LIN {X -0.049,Y -176.502,Z 1174.767,A 0.000,B 0.000,C 90.000,E1 138.162} C_DIS
LIN {X 0.075,Y -180.801,Z 1174.753,A 0.000,B 0.000,C 90.000,E1 135.567} C_DIS
LIN {X 0.061,Y -186.209,Z 1174.735,A 0.000,B 0.000,C 90.000,E1 132.204} C_DIS
LIN {X 0.000,Y -190.846,Z 1174.721,A 0.000,B 0.000,C 90.000,E1 129.725} C_DIS
LIN {X 0.034,Y -196.606,Z 1174.702,A 0.000,B 0.000,C 90.000,E1 126.423} C_DIS
LIN {X 0.006,Y -201.153,Z 1174.690,A 0.000,B 0.000,C 90.000,E1 124.119} C_DIS
LIN {X -0.026,Y -310.936,Z 1174.690,A 0.000,B 0.000,C 90.000,E1 124.119} C_DIS
LIN {X 0.002,Y -315.080,Z 1174.689,A 0.000,B 0.000,C 90.000,E1 123.992} C_DIS
LIN {X 0.113,Y -317.999,Z 1174.688,A 0.000,B 0.000,C 90.000,E1 123.785} C_DIS
LIN {X 0.000,Y -321.723,Z 1174.686,A 0.000,B 0.000,C 90.000,E1 123.420} C_DIS
LIN {X 0.084,Y -325.167,Z 1174.682,A 0.000,B 0.000,C 90.000,E1 122.832} C_DIS
LIN {X -0.013,Y -327.638,Z 1174.679,A 0.000,B 0.000,C 90.000,E1 122.212} C_DIS
LIN {X -0.136,Y -338.542,Z 1174.663,A 0.000,B 0.000,C 90.000,E1 119.411} C_DIS
LIN {X 0.016,Y -350.831,Z 1174.648,A 0.000,B 0.000,C 90.000,E1 116.616} C_DIS
LIN {X 0.063,Y -364.604,Z 1174.633,A 0.000,B 0.000,C 90.000,E1 113.898} C_DIS
LIN {X 0.100,Y -378.196,Z 1174.620,A 0.000,B 0.000,C 90.000,E1 111.535} C_DIS
LIN {X -0.165,Y -393.156,Z 1174.607,A 0.000,B 0.000,C 90.000,E1 109.268} C_DIS
LIN {X 0.055,Y -409.587,Z 1174.594,A 0.000,B 0.000,C 90.000,E1 106.985} C_DIS
LIN {X 0.182,Y -427.609,Z 1174.582,A 0.000,B 0.000,C 90.000,E1 104.773} C_DIS
LIN {X 0.246,Y -447.177,Z 1174.570,A 0.000,B 0.000,C 90.000,E1 102.647} C_DIS
LIN {X -0.025,Y -470.021,Z 1174.558,A 0.000,B 0.000,C 90.000,E1 100.489} C_DIS
LIN {X -0.016,Y -472.082,Z 1174.557,A 0.000,B 0.000,C 90.000,E1 100.254} C_DIS
LIN {X -0.007,Y -473.647,Z 1174.556,A 0.000,B 0.000,C 90.000,E1 100.018} C_DIS
LIN {X -0.147,Y -474.925,Z 1174.554,A 0.000,B 0.000,C 90.000,E1 99.782} C_DIS
LIN {X 0.101,Y -475.866,Z 1174.553,A 0.000,B 0.000,C 90.000,E1 99.500} C_DIS
LIN {X -0.166,Y -476.904,Z 1174.550,A 0.000,B 0.000,C 90.000,E1 99.029} C_DIS
LIN {X -0.033,Y -476.952,Z 1174.547,A 0.000,B 0.000,C 90.000,E1 98.511} C_DIS
LIN {X 0.109,Y -476.021,Z 1174.544,A 0.000,B 0.000,C 90.000,E1 97.992} C_DIS
LIN {X -0.219,Y -473.955,Z 1174.542,A 0.000,B 0.000,C 90.000,E1 97.530} C_DIS
LIN {X 0.115,Y -472.362,Z 1174.540,A 0.000,B 0.000,C 90.000,E1 97.239} C_DIS
LIN {X 0.027,Y -457.874,Z 1174.529,A 0.000,B 0.000,C 90.000,E1 95.220} C_DIS
LIN {X -0.055,Y -440.340,Z 1174.515,A 0.000,B 0.000,C 90.000,E1 92.636} C_DIS
LIN {X -0.091,Y -422.563,Z 1174.498,A 0.000,B 0.000,C 90.000,E1 89.714} C_DIS
LIN {X -0.002,Y -409.192,Z 1174.485,A 0.000,B 0.000,C 90.000,E1 87.249} C_DIS
LIN {X 0.069,Y -398.908,Z 1174.474,A 0.000,B 0.000,C 90.000,E1 85.298} C_DIS
LIN {X 0.035,Y -385.631,Z 1174.460,A 0.000,B 0.000,C 90.000,E1 82.761} C_DIS
LIN {X 0.104,Y -376.810,Z 1174.450,A 0.000,B 0.000,C 90.000,E1 81.027} C_DIS
LIN {X 0.065,Y -367.674,Z 1174.441,A 0.000,B 0.000,C 90.000,E1 79.285} C_DIS
LIN {X 0.006,Y -358.241,Z 1174.431,A 0.000,B 0.000,C 90.000,E1 77.521} C_DIS
LIN {X 0.129,Y -348.588,Z 1174.421,A 0.000,B 0.000,C 90.000,E1 75.700} C_DIS
LIN {X 0.145,Y -337.276,Z 1174.409,A 0.000,B 0.000,C 90.000,E1 73.559} C_DIS
LIN {X -0.024,Y -324.592,Z 1174.395,A 0.000,B 0.000,C 90.000,E1 71.094} C_DIS
LIN {X -0.063,Y -310.987,Z 1174.379,A 0.000,B 0.000,C 90.000,E1 68.230} C_DIS
LIN {X -0.001,Y -298.149,Z 1174.363,A 0.000,B 0.000,C 90.000,E1 65.281} C_DIS
LIN {X -0.038,Y -286.076,Z 1174.346,A 0.000,B 0.000,C 90.000,E1 62.281} C_DIS
LIN {X -0.066,Y -273.394,Z 1174.327,A 0.000,B 0.000,C 90.000,E1 58.869} C_DIS
LIN {X -0.117,Y -263.733,Z 1174.311,A 0.000,B 0.000,C 90.000,E1 56.087} C_DIS
LIN {X 0.091,Y -252.281,Z 1174.292,A 0.000,B 0.000,C 90.000,E1 52.477} C_DIS
LIN {X 0.027,Y -242.627,Z 1174.273,A 0.000,B 0.000,C 90.000,E1 49.218} C_DIS
LIN {X 0.132,Y -232.705,Z 1174.253,A 0.000,B 0.000,C 90.000,E1 45.486} C_DIS
LIN {X -0.074,Y -223.677,Z 1174.232,A 0.000,B 0.000,C 90.000,E1 41.757} C_DIS
LIN {X -0.011,Y -215.431,Z 1174.210,A 0.000,B 0.000,C 90.000,E1 37.890} C_DIS
LIN {X -0.081,Y -207.948,Z 1174.189,A 0.000,B 0.000,C 90.000,E1 33.992} C_DIS
LIN {X -0.038,Y -201.142,Z 1174.167,A 0.000,B 0.000,C 90.000,E1 30.001} C_DIS
LIN {X -0.083,Y -195.095,Z 1174.144,A 0.000,B 0.000,C 90.000,E1 25.976} C_DIS
LIN {X 0.054,Y -189.968,Z 1174.121,A 0.000,B 0.000,C 90.000,E1 21.844} C_DIS
LIN {X 0.099,Y -185.676,Z 1174.099,A 0.000,B 0.000,C 90.000,E1 17.692} C_DIS
LIN {X 0.036,Y -182.382,Z 1174.075,A 0.000,B 0.000,C 90.000,E1 13.536} C_DIS
LIN {X 0.030,Y -179.396,Z 1174.042,A 0.000,B 0.000,C 90.000,E1 7.644} C_DIS
LIN {X 0.062,Y -180.217,Z 1173.969,A 0.000,B 0.000,C 90.000,E1 354.432} C_DIS
LIN {X -0.014,Y -183.167,Z 1173.941,A 0.000,B 0.000,C 90.000,E1 349.398} C_DIS
LIN {X -0.066,Y -186.673,Z 1173.918,A 0.000,B 0.000,C 90.000,E1 345.227} C_DIS
LIN {X 0.052,Y -191.138,Z 1173.895,A 0.000,B 0.000,C 90.000,E1 341.040} C_DIS
LIN {X 0.086,Y -196.284,Z 1173.872,A 0.000,B 0.000,C 90.000,E1 336.922} C_DIS
LIN {X 0.053,Y -202.230,Z 1173.849,A 0.000,B 0.000,C 90.000,E1 332.871} C_DIS
LIN {X 0.040,Y -208.789,Z 1173.827,A 0.000,B 0.000,C 90.000,E1 328.869} C_DIS
LIN {X 0.135,Y -215.942,Z 1173.805,A 0.000,B 0.000,C 90.000,E1 324.895} C_DIS
LIN {X -0.029,Y -222.299,Z 1173.788,A 0.000,B 0.000,C 90.000,E1 321.823} C_DIS
LIN {X -0.113,Y -229.684,Z 1173.771,A 0.000,B 0.000,C 90.000,E1 318.771} C_DIS
LIN {X 0.104,Y -239.207,Z 1173.752,A 0.000,B 0.000,C 90.000,E1 315.324} C_DIS
LIN {X 0.104,Y -250.116,Z 1173.734,A 0.000,B 0.000,C 90.000,E1 312.000} C_DIS
LIN {X 0.109,Y -262.391,Z 1173.715,A 0.000,B 0.000,C 90.000,E1 308.749} C_DIS
LIN {X -0.068,Y -271.258,Z 1173.704,A 0.000,B 0.000,C 90.000,E1 306.664} C_DIS
LIN {X 0.145,Y -280.911,Z 1173.692,A 0.000,B 0.000,C 90.000,E1 304.532} C_DIS
LIN {X 0.075,Y -291.557,Z 1173.681,A 0.000,B 0.000,C 90.000,E1 302.498} C_DIS
LIN {X -0.160,Y -307.099,Z 1173.666,A 0.000,B 0.000,C 90.000,E1 299.873} C_DIS
LIN {X -0.040,Y -319.840,Z 1173.655,A 0.000,B 0.000,C 90.000,E1 297.897} C_DIS
LIN {X 0.071,Y -331.588,Z 1173.646,A 0.000,B 0.000,C 90.000,E1 296.283} C_DIS
LIN {X -0.064,Y -354.903,Z 1173.631,A 0.000,B 0.000,C 90.000,E1 293.567} C_DIS
LIN {X -0.085,Y -370.931,Z 1173.622,A 0.000,B 0.000,C 90.000,E1 291.897} C_DIS
LIN {X 0.197,Y -392.686,Z 1173.610,A 0.000,B 0.000,C 90.000,E1 289.812} C_DIS
LIN {X -0.061,Y -403.296,Z 1173.605,A 0.000,B 0.000,C 90.000,E1 288.852} C_DIS
LIN {X -0.119,Y -411.028,Z 1173.600,A 0.000,B 0.000,C 90.000,E1 288.109} C_DIS
LIN {X 0.117,Y -421.163,Z 1173.595,A 0.000,B 0.000,C 90.000,E1 287.040} C_DIS
LIN {X -0.004,Y -428.577,Z 1173.590,A 0.000,B 0.000,C 90.000,E1 286.260} C_DIS
LIN {X 0.222,Y -435.639,Z 1173.586,A 0.000,B 0.000,C 90.000,E1 285.426} C_DIS
LIN {X -0.038,Y -442.111,Z 1173.581,A 0.000,B 0.000,C 90.000,E1 284.662} C_DIS
LIN {X -0.141,Y -447.808,Z 1173.577,A 0.000,B 0.000,C 90.000,E1 283.883} C_DIS
LIN {X 0.141,Y -452.846,Z 1173.573,A 0.000,B 0.000,C 90.000,E1 283.063} C_DIS
LIN {X 0.025,Y -457.271,Z 1173.568,A 0.000,B 0.000,C 90.000,E1 282.299} C_DIS
LIN {X -0.050,Y -461.054,Z 1173.564,A 0.000,B 0.000,C 90.000,E1 281.535} C_DIS
LIN {X -0.188,Y -464.245,Z 1173.560,A 0.000,B 0.000,C 90.000,E1 280.782} C_DIS
LIN {X -0.051,Y -466.130,Z 1173.557,A 0.000,B 0.000,C 90.000,E1 280.254} C_DIS
LIN {X 0.089,Y -467.783,Z 1173.554,A 0.000,B 0.000,C 90.000,E1 279.726} C_DIS
LIN {X 0.163,Y -469.229,Z 1173.551,A 0.000,B 0.000,C 90.000,E1 279.208} C_DIS
LIN {X -0.216,Y -470.449,Z 1173.548,A 0.000,B 0.000,C 90.000,E1 278.746} C_DIS
LIN {X -0.051,Y -471.453,Z 1173.546,A 0.000,B 0.000,C 90.000,E1 278.219} C_DIS
LIN {X 0.053,Y -472.097,Z 1173.543,A 0.000,B 0.000,C 90.000,E1 277.701} C_DIS
LIN {X 0.163,Y -472.368,Z 1173.540,A 0.000,B 0.000,C 90.000,E1 277.182} C_DIS
LIN {X -0.191,Y -472.233,Z 1173.537,A 0.000,B 0.000,C 90.000,E1 276.720} C_DIS
LIN {X -0.073,Y -471.696,Z 1173.534,A 0.000,B 0.000,C 90.000,E1 276.201} C_DIS
LIN {X 0.043,Y -470.719,Z 1173.532,A 0.000,B 0.000,C 90.000,E1 275.682} C_DIS
LIN {X 0.155,Y -469.304,Z 1173.529,A 0.000,B 0.000,C 90.000,E1 275.163} C_DIS
LIN {X -0.208,Y -467.421,Z 1173.526,A 0.000,B 0.000,C 90.000,E1 274.702} C_DIS
LIN {X -0.149,Y -465.013,Z 1173.523,A 0.000,B 0.000,C 90.000,E1 274.188} C_DIS
LIN {X -0.071,Y -461.983,Z 1173.520,A 0.000,B 0.000,C 90.000,E1 273.669} C_DIS
LIN {X -0.039,Y -458.095,Z 1173.517,A 0.000,B 0.000,C 90.000,E1 273.154} C_DIS
LIN {X 0.220,Y -455.772,Z 1173.516,A 0.000,B 0.000,C 90.000,E1 272.865} C_DIS
LIN {X -0.138,Y -450.334,Z 1173.513,A 0.000,B 0.000,C 90.000,E1 272.407} C_DIS
LIN {X -0.112,Y -444.074,Z 1173.511,A 0.000,B 0.000,C 90.000,E1 271.949} C_DIS
LIN {X 0.025,Y -437.430,Z 1173.509,A 0.000,B 0.000,C 90.000,E1 271.547} C_DIS
LIN {X 0.201,Y -430.402,Z 1173.507,A 0.000,B 0.000,C 90.000,E1 271.203} C_DIS
LIN {X -0.067,Y -423.443,Z 1173.505,A 0.000,B 0.000,C 90.000,E1 270.974} C_DIS
LIN {X -0.032,Y -416.454,Z 1173.504,A 0.000,B 0.000,C 90.000,E1 270.745} C_DIS
LIN {X 0.056,Y -405.575,Z 1173.503,A 0.000,B 0.000,C 90.000,E1 270.458} C_DIS
LIN {X 0.138,Y -391.567,Z 1173.501,A 0.000,B 0.000,C 90.000,E1 270.172} C_DIS
LIN {X 0.102,Y -383.629,Z 1173.500,A 0.000,B 0.000,C 90.000,E1 270.057} C_DIS
LIN {X -0.178,Y -371.294,Z 1173.500,A 0.000,B 0.000,C 90.000,E1 270.000} C_DIS
LIN {X 0.140,Y -369.390,Z 1173.500,A 0.000,B 0.000,C 90.000,E1 269.943} C_DIS
LIN {X 0.044,Y -181.553,Z 1173.500,A 0.000,B 0.000,C 90.000,E1 269.943} C_DIS
LIN {X 0.055,Y -180.823,Z 1173.471,A 0.000,B 0.000,C 90.000,E1 264.837} C_DIS
LIN {X -0.044,Y -178.926,Z 1173.443,A 0.000,B 0.000,C 90.000,E1 259.803} C_DIS
LIN {X -0.006,Y -175.974,Z 1173.415,A 0.000,B 0.000,C 90.000,E1 254.700} C_DIS
LIN {X -0.061,Y -175.460,Z 1173.410,A 0.000,B 0.000,C 90.000,E1 253.866} C_DIS
LIN {X -0.004,Y -172.211,Z 1173.386,A 0.000,B 0.000,C 90.000,E1 249.571} C_DIS
LIN {X -0.026,Y -171.686,Z 1173.382,A 0.000,B 0.000,C 90.000,E1 248.720} C_DIS
LIN {X -0.035,Y -167.913,Z 1173.358,A 0.000,B 0.000,C 90.000,E1 244.409} C_DIS
LIN {X -0.017,Y -166.655,Z 1173.348,A 0.000,B 0.000,C 90.000,E1 242.666} C_DIS
LIN {X 0.038,Y -162.638,Z 1173.324,A 0.000,B 0.000,C 90.000,E1 238.280} C_DIS
LIN {X -0.038,Y -161.326,Z 1173.314,A 0.000,B 0.000,C 90.000,E1 236.548} C_DIS
LIN {X 0.005,Y -157.322,Z 1173.290,A 0.000,B 0.000,C 90.000,E1 232.110} C_DIS
LIN {X -0.062,Y -155.303,Z 1173.275,A 0.000,B 0.000,C 90.000,E1 229.461} C_DIS
LIN {X 0.084,Y -151.662,Z 1173.250,A 0.000,B 0.000,C 90.000,E1 224.919} C_DIS
LIN {X 0.021,Y -150.529,Z 1173.240,A 0.000,B 0.000,C 90.000,E1 223.137} C_DIS
LIN {X -0.048,Y -147.253,Z 1173.214,A 0.000,B 0.000,C 90.000,E1 218.624} C_DIS
LIN {X 0.008,Y -145.278,Z 1173.194,A 0.000,B 0.000,C 90.000,E1 214.945} C_DIS
LIN {X 0.042,Y -142.382,Z 1173.163,A 0.000,B 0.000,C 90.000,E1 209.411} C_DIS
LIN {X -0.035,Y -141.359,Z 1173.148,A 0.000,B 0.000,C 90.000,E1 206.668} C_DIS
LIN {X 0.074,Y -139.342,Z 1173.112,A 0.000,B 0.000,C 90.000,E1 200.120} C_DIS
LIN {X -0.051,Y -139.010,Z 1173.102,A 0.000,B 0.000,C 90.000,E1 198.308} C_DIS
LIN {X -0.056,Y -138.341,Z 1173.055,A 0.000,B 0.000,C 90.000,E1 189.905} C_DIS
LIN {X -0.036,Y -139.399,Z 1173.008,A 0.000,B 0.000,C 90.000,E1 181.489} C_DIS
LIN {X 0.017,Y -141.304,Z 1172.972,A 0.000,B 0.000,C 90.000,E1 174.951} C_DIS
LIN {X -0.025,Y -142.664,Z 1172.957,A 0.000,B 0.000,C 90.000,E1 172.186} C_DIS
LIN {X -0.076,Y -145.011,Z 1172.931,A 0.000,B 0.000,C 90.000,E1 167.589} C_DIS
LIN {X 0.055,Y -147.638,Z 1172.911,A 0.000,B 0.000,C 90.000,E1 163.866} C_DIS
LIN {X -0.009,Y -150.270,Z 1172.890,A 0.000,B 0.000,C 90.000,E1 160.242} C_DIS
LIN {X 0.004,Y -153.671,Z 1172.870,A 0.000,B 0.000,C 90.000,E1 156.613} C_DIS
LIN {X 0.061,Y -157.086,Z 1172.850,A 0.000,B 0.000,C 90.000,E1 152.999} C_DIS
LIN {X -0.002,Y -161.221,Z 1172.830,A 0.000,B 0.000,C 90.000,E1 149.459} C_DIS
LIN {X -0.054,Y -163.310,Z 1172.821,A 0.000,B 0.000,C 90.000,E1 147.709} C_DIS
LIN {X -0.044,Y -167.760,Z 1172.801,A 0.000,B 0.000,C 90.000,E1 144.196} C_DIS
LIN {X 0.108,Y -171.576,Z 1172.786,A 0.000,B 0.000,C 90.000,E1 141.537} C_DIS
LIN {X -0.092,Y -176.525,Z 1172.767,A 0.000,B 0.000,C 90.000,E1 138.162} C_DIS
LIN {X 0.032,Y -180.823,Z 1172.753,A 0.000,B 0.000,C 90.000,E1 135.567} C_DIS
LIN {X 0.017,Y -186.232,Z 1172.734,A 0.000,B 0.000,C 90.000,E1 132.204} C_DIS
LIN {X -0.045,Y -190.869,Z 1172.721,A 0.000,B 0.000,C 90.000,E1 129.725} C_DIS
LIN {X -0.012,Y -196.631,Z 1172.702,A 0.000,B 0.000,C 90.000,E1 126.423} C_DIS
LIN {X 0.079,Y -201.118,Z 1172.690,A 0.000,B 0.000,C 90.000,E1 124.119} C_DIS
LIN {X 0.086,Y -310.102,Z 1172.690,A 0.000,B 0.000,C 90.000,E1 124.119} C_DIS
LIN {X -0.070,Y -315.565,Z 1172.689,A 0.000,B 0.000,C 90.000,E1 123.992} C_DIS
LIN {X -0.063,Y -318.498,Z 1172.688,A 0.000,B 0.000,C 90.000,E1 123.785} C_DIS
LIN {X -0.088,Y -322.233,Z 1172.685,A 0.000,B 0.000,C 90.000,E1 123.372} C_DIS
LIN {X 0.086,Y -324.120,Z 1172.684,A 0.000,B 0.000,C 90.000,E1 123.038} C_DIS
LIN {X -0.013,Y -325.596,Z 1172.682,A 0.000,B 0.000,C 90.000,E1 122.752} C_DIS
LIN {X 0.078,Y -338.901,Z 1172.663,A 0.000,B 0.000,C 90.000,E1 119.283} C_DIS
LIN {X -0.065,Y -351.237,Z 1172.647,A 0.000,B 0.000,C 90.000,E1 116.539} C_DIS
LIN {X -0.018,Y -365.061,Z 1172.632,A 0.000,B 0.000,C 90.000,E1 113.823} C_DIS
LIN {X 0.020,Y -378.702,Z 1172.619,A 0.000,B 0.000,C 90.000,E1 111.461} C_DIS
LIN {X 0.126,Y -393.714,Z 1172.606,A 0.000,B 0.000,C 90.000,E1 109.141} C_DIS
LIN {X -0.024,Y -410.202,Z 1172.594,A 0.000,B 0.000,C 90.000,E1 106.913} C_DIS
LIN {X -0.005,Y -428.284,Z 1172.582,A 0.000,B 0.000,C 90.000,E1 104.717} C_DIS
LIN {X 0.092,Y -447.891,Z 1172.570,A 0.000,B 0.000,C 90.000,E1 102.591} C_DIS
LIN {X -0.043,Y -470.651,Z 1172.558,A 0.000,B 0.000,C 90.000,E1 100.423} C_DIS
LIN {X -0.166,Y -472.574,Z 1172.557,A 0.000,B 0.000,C 90.000,E1 100.197} C_DIS
LIN {X -0.204,Y -474.036,Z 1172.555,A 0.000,B 0.000,C 90.000,E1 99.962} C_DIS
LIN {X -0.093,Y -476.032,Z 1172.552,A 0.000,B 0.000,C 90.000,E1 99.443} C_DIS
LIN {X 0.106,Y -476.898,Z 1172.550,A 0.000,B 0.000,C 90.000,E1 98.916} C_DIS
LIN {X -0.230,Y -476.784,Z 1172.547,A 0.000,B 0.000,C 90.000,E1 98.454} C_DIS
LIN {X -0.088,Y -475.679,Z 1172.544,A 0.000,B 0.000,C 90.000,E1 97.936} C_DIS
LIN {X -0.219,Y -474.704,Z 1172.543,A 0.000,B 0.000,C 90.000,E1 97.701} C_DIS
LIN {X 0.118,Y -473.387,Z 1172.541,A 0.000,B 0.000,C 90.000,E1 97.409} C_DIS
LIN {X 0.045,Y -458.988,Z 1172.530,A 0.000,B 0.000,C 90.000,E1 95.391} C_DIS
LIN {X -0.012,Y -441.392,Z 1172.516,A 0.000,B 0.000,C 90.000,E1 92.808} C_DIS
LIN {X 0.103,Y -421.988,Z 1172.498,A 0.000,B 0.000,C 90.000,E1 89.599} C_DIS
LIN {X 0.170,Y -408.639,Z 1172.484,A 0.000,B 0.000,C 90.000,E1 87.135} C_DIS
LIN {X -0.174,Y -398.345,Z 1172.473,A 0.000,B 0.000,C 90.000,E1 85.241} C_DIS
LIN {X 0.166,Y -385.048,Z 1172.459,A 0.000,B 0.000,C 90.000,E1 82.648} C_DIS
LIN {X -0.154,Y -376.199,Z 1172.450,A 0.000,B 0.000,C 90.000,E1 80.971} C_DIS
LIN {X -0.130,Y -367.052,Z 1172.440,A 0.000,B 0.000,C 90.000,E1 79.218} C_DIS
LIN {X 0.085,Y -357.601,Z 1172.430,A 0.000,B 0.000,C 90.000,E1 77.409} C_DIS
LIN {X -0.149,Y -347.926,Z 1172.420,A 0.000,B 0.000,C 90.000,E1 75.644} C_DIS
LIN {X 0.167,Y -334.992,Z 1172.406,A 0.000,B 0.000,C 90.000,E1 73.142} C_DIS
LIN {X -0.059,Y -322.397,Z 1172.393,A 0.000,B 0.000,C 90.000,E1 70.678} C_DIS
LIN {X 0.183,Y -306.046,Z 1172.373,A 0.000,B 0.000,C 90.000,E1 67.102} C_DIS
LIN {X -0.031,Y -292.134,Z 1172.355,A 0.000,B 0.000,C 90.000,E1 63.845} C_DIS
LIN {X 0.019,Y -280.314,Z 1172.338,A 0.000,B 0.000,C 90.000,E1 60.795} C_DIS
LIN {X -0.072,Y -269.159,Z 1172.321,A 0.000,B 0.000,C 90.000,E1 57.709} C_DIS
LIN {X -0.033,Y -258.483,Z 1172.303,A 0.000,B 0.000,C 90.000,E1 54.529} C_DIS
LIN {X -0.045,Y -248.425,Z 1172.285,A 0.000,B 0.000,C 90.000,E1 51.295} C_DIS
LIN {X -0.059,Y -238.057,Z 1172.265,A 0.000,B 0.000,C 90.000,E1 47.634} C_DIS
LIN {X 0.055,Y -228.506,Z 1172.244,A 0.000,B 0.000,C 90.000,E1 43.866} C_DIS
LIN {X -0.097,Y -219.812,Z 1172.223,A 0.000,B 0.000,C 90.000,E1 40.092} C_DIS
LIN {X 0.052,Y -211.901,Z 1172.201,A 0.000,B 0.000,C 90.000,E1 36.171} C_DIS
LIN {X 0.092,Y -204.686,Z 1172.179,A 0.000,B 0.000,C 90.000,E1 32.212} C_DIS
LIN {X -0.005,Y -198.166,Z 1172.157,A 0.000,B 0.000,C 90.000,E1 28.231} C_DIS
LIN {X 0.035,Y -192.459,Z 1172.134,A 0.000,B 0.000,C 90.000,E1 24.155} C_DIS
LIN {X -0.053,Y -187.661,Z 1172.111,A 0.000,B 0.000,C 90.000,E1 20.066} C_DIS
LIN {X -0.020,Y -183.796,Z 1172.088,A 0.000,B 0.000,C 90.000,E1 15.898} C_DIS
LIN {X 0.062,Y -180.484,Z 1172.060,A 0.000,B 0.000,C 90.000,E1 10.838} C_DIS
LIN {X 0.063,Y -178.329,Z 1172.023,A 0.000,B 0.000,C 90.000,E1 4.073} C_DIS
LIN {X 0.050,Y -179.888,Z 1171.969,A 0.000,B 0.000,C 90.000,E1 354.432} C_DIS
LIN {X -0.038,Y -182.831,Z 1171.941,A 0.000,B 0.000,C 90.000,E1 349.398} C_DIS
LIN {X 0.079,Y -186.309,Z 1171.918,A 0.000,B 0.000,C 90.000,E1 345.172} C_DIS
LIN {X 0.004,Y -190.771,Z 1171.895,A 0.000,B 0.000,C 90.000,E1 341.040} C_DIS
LIN {X 0.024,Y -195.923,Z 1171.872,A 0.000,B 0.000,C 90.000,E1 336.922} C_DIS
LIN {X -0.020,Y -201.848,Z 1171.849,A 0.000,B 0.000,C 90.000,E1 332.871} C_DIS
LIN {X -0.050,Y -208.422,Z 1171.827,A 0.000,B 0.000,C 90.000,E1 328.869} C_DIS
LIN {X 0.031,Y -215.610,Z 1171.805,A 0.000,B 0.000,C 90.000,E1 324.895} C_DIS
LIN {X 0.030,Y -222.026,Z 1171.788,A 0.000,B 0.000,C 90.000,E1 321.778} C_DIS
LIN {X 0.086,Y -229.469,Z 1171.771,A 0.000,B 0.000,C 90.000,E1 318.690} C_DIS
LIN {X -0.033,Y -239.035,Z 1171.752,A 0.000,B 0.000,C 90.000,E1 315.324} C_DIS
LIN {X -0.044,Y -249.981,Z 1171.733,A 0.000,B 0.000,C 90.000,E1 312.000} C_DIS
LIN {X -0.050,Y -262.317,Z 1171.715,A 0.000,B 0.000,C 90.000,E1 308.749} C_DIS
LIN {X 0.146,Y -271.213,Z 1171.703,A 0.000,B 0.000,C 90.000,E1 306.583} C_DIS
LIN {X -0.083,Y -282.636,Z 1171.690,A 0.000,B 0.000,C 90.000,E1 304.199} C_DIS
LIN {X 0.032,Y -293.524,Z 1171.679,A 0.000,B 0.000,C 90.000,E1 302.133} C_DIS
LIN {X 0.074,Y -307.185,Z 1171.666,A 0.000,B 0.000,C 90.000,E1 299.795} C_DIS
LIN {X 0.052,Y -319.953,Z 1171.655,A 0.000,B 0.000,C 90.000,E1 297.847} C_DIS
LIN {X 0.172,Y -331.725,Z 1171.646,A 0.000,B 0.000,C 90.000,E1 296.232} C_DIS
LIN {X 0.092,Y -352.148,Z 1171.632,A 0.000,B 0.000,C 90.000,E1 293.823} C_DIS
LIN {X 0.011,Y -367.983,Z 1171.623,A 0.000,B 0.000,C 90.000,E1 292.153} C_DIS
LIN {X -0.135,Y -389.737,Z 1171.612,A 0.000,B 0.000,C 90.000,E1 290.120} C_DIS
LIN {X 0.151,Y -400.402,Z 1171.606,A 0.000,B 0.000,C 90.000,E1 289.087} C_DIS
LIN {X -0.083,Y -408.312,Z 1171.602,A 0.000,B 0.000,C 90.000,E1 288.362} C_DIS
LIN {X -0.057,Y -418.508,Z 1171.596,A 0.000,B 0.000,C 90.000,E1 287.330} C_DIS
LIN {X 0.051,Y -428.488,Z 1171.590,A 0.000,B 0.000,C 90.000,E1 286.260} C_DIS
LIN {X -0.141,Y -435.570,Z 1171.586,A 0.000,B 0.000,C 90.000,E1 285.481} C_DIS
LIN {X 0.019,Y -442.041,Z 1171.581,A 0.000,B 0.000,C 90.000,E1 284.662} C_DIS
LIN {X -0.085,Y -447.763,Z 1171.577,A 0.000,B 0.000,C 90.000,E1 283.883} C_DIS
LIN {X 0.198,Y -452.808,Z 1171.573,A 0.000,B 0.000,C 90.000,E1 283.063} C_DIS
LIN {X 0.081,Y -457.266,Z 1171.568,A 0.000,B 0.000,C 90.000,E1 282.299} C_DIS
LIN {X 0.007,Y -461.060,Z 1171.564,A 0.000,B 0.000,C 90.000,E1 281.535} C_DIS
LIN {X -0.131,Y -464.245,Z 1171.560,A 0.000,B 0.000,C 90.000,E1 280.782} C_DIS
LIN {X 0.007,Y -466.155,Z 1171.557,A 0.000,B 0.000,C 90.000,E1 280.254} C_DIS
LIN {X 0.147,Y -467.851,Z 1171.554,A 0.000,B 0.000,C 90.000,E1 279.726} C_DIS
LIN {X 0.221,Y -469.332,Z 1171.551,A 0.000,B 0.000,C 90.000,E1 279.208} C_DIS
LIN {X -0.156,Y -470.596,Z 1171.548,A 0.000,B 0.000,C 90.000,E1 278.746} C_DIS
LIN {X 0.009,Y -471.575,Z 1171.546,A 0.000,B 0.000,C 90.000,E1 278.219} C_DIS
LIN {X 0.113,Y -472.242,Z 1171.543,A 0.000,B 0.000,C 90.000,E1 277.701} C_DIS
LIN {X 0.225,Y -472.567,Z 1171.540,A 0.000,B 0.000,C 90.000,E1 277.182} C_DIS
LIN {X -0.128,Y -472.452,Z 1171.537,A 0.000,B 0.000,C 90.000,E1 276.720} C_DIS
LIN {X -0.010,Y -471.944,Z 1171.534,A 0.000,B 0.000,C 90.000,E1 276.201} C_DIS
LIN {X 0.107,Y -471.007,Z 1171.532,A 0.000,B 0.000,C 90.000,E1 275.682} C_DIS
LIN {X 0.220,Y -469.624,Z 1171.529,A 0.000,B 0.000,C 90.000,E1 275.163} C_DIS
LIN {X -0.142,Y -467.798,Z 1171.526,A 0.000,B 0.000,C 90.000,E1 274.702} C_DIS
LIN {X -0.080,Y -465.391,Z 1171.523,A 0.000,B 0.000,C 90.000,E1 274.188} C_DIS
LIN {X 0.000,Y -462.390,Z 1171.520,A 0.000,B 0.000,C 90.000,E1 273.669} C_DIS
LIN {X 0.034,Y -458.543,Z 1171.518,A 0.000,B 0.000,C 90.000,E1 273.154} C_DIS
LIN {X -0.163,Y -456.262,Z 1171.516,A 0.000,B 0.000,C 90.000,E1 272.922} C_DIS
LIN {X 0.073,Y -453.668,Z 1171.515,A 0.000,B 0.000,C 90.000,E1 272.636} C_DIS
LIN {X -0.084,Y -450.819,Z 1171.513,A 0.000,B 0.000,C 90.000,E1 272.407} C_DIS
LIN {X -0.109,Y -444.586,Z 1171.511,A 0.000,B 0.000,C 90.000,E1 271.949} C_DIS
LIN {X -0.022,Y -437.865,Z 1171.509,A 0.000,B 0.000,C 90.000,E1 271.547} C_DIS
LIN {X 0.119,Y -430.822,Z 1171.507,A 0.000,B 0.000,C 90.000,E1 271.203} C_DIS
LIN {X -0.163,Y -423.858,Z 1171.505,A 0.000,B 0.000,C 90.000,E1 270.974} C_DIS
LIN {X -0.112,Y -416.957,Z 1171.504,A 0.000,B 0.000,C 90.000,E1 270.745} C_DIS
LIN {X 0.188,Y -409.846,Z 1171.503,A 0.000,B 0.000,C 90.000,E1 270.516} C_DIS
LIN {X 0.174,Y -399.186,Z 1171.502,A 0.000,B 0.000,C 90.000,E1 270.286} C_DIS
LIN {X 0.049,Y -388.425,Z 1171.501,A 0.000,B 0.000,C 90.000,E1 270.115} C_DIS
LIN {X 0.083,Y -379.778,Z 1171.500,A 0.000,B 0.000,C 90.000,E1 270.000} C_DIS
LIN {X 0.080,Y -371.038,Z 1171.500,A 0.000,B 0.000,C 90.000,E1 269.943} C_DIS
LIN {X 0.026,Y -365.401,Z 1171.500,A 0.000,B 0.000,C 90.000,E1 269.943} C_DIS
LIN {X -0.013,Y -181.550,Z 1171.500,A 0.000,B 0.000,C 90.000,E1 269.943} C_DIS
LIN {X 0.021,Y -180.819,Z 1171.471,A 0.000,B 0.000,C 90.000,E1 264.837} C_DIS
LIN {X -0.078,Y -178.922,Z 1171.443,A 0.000,B 0.000,C 90.000,E1 259.803} C_DIS
LIN {X 0.006,Y -175.969,Z 1171.415,A 0.000,B 0.000,C 90.000,E1 254.685} C_DIS
LIN {X -0.046,Y -175.451,Z 1171.410,A 0.000,B 0.000,C 90.000,E1 253.850} C_DIS
LIN {X -0.037,Y -172.204,Z 1171.386,A 0.000,B 0.000,C 90.000,E1 249.571} C_DIS
LIN {X -0.059,Y -171.679,Z 1171.382,A 0.000,B 0.000,C 90.000,E1 248.720} C_DIS
LIN {X -0.068,Y -167.904,Z 1171.358,A 0.000,B 0.000,C 90.000,E1 244.409} C_DIS
LIN {X -0.050,Y -166.645,Z 1171.348,A 0.000,B 0.000,C 90.000,E1 242.666} C_DIS
LIN {X 0.005,Y -162.630,Z 1171.324,A 0.000,B 0.000,C 90.000,E1 238.280} C_DIS
LIN {X 0.064,Y -161.317,Z 1171.314,A 0.000,B 0.000,C 90.000,E1 236.501} C_DIS
LIN {X -0.026,Y -157.313,Z 1171.289,A 0.000,B 0.000,C 90.000,E1 232.110} C_DIS
LIN {X -0.093,Y -155.291,Z 1171.275,A 0.000,B 0.000,C 90.000,E1 229.461} C_DIS
LIN {X 0.053,Y -151.653,Z 1171.250,A 0.000,B 0.000,C 90.000,E1 224.919} C_DIS
LIN {X -0.010,Y -150.520,Z 1171.240,A 0.000,B 0.000,C 90.000,E1 223.137} C_DIS
LIN {X 0.014,Y -147.246,Z 1171.214,A 0.000,B 0.000,C 90.000,E1 218.588} C_DIS
LIN {X -0.022,Y -145.271,Z 1171.194,A 0.000,B 0.000,C 90.000,E1 214.945} C_DIS
LIN {X 0.012,Y -142.378,Z 1171.163,A 0.000,B 0.000,C 90.000,E1 209.411} C_DIS
LIN {X 0.062,Y -141.354,Z 1171.148,A 0.000,B 0.000,C 90.000,E1 206.616} C_DIS
LIN {X 0.045,Y -139.340,Z 1171.112,A 0.000,B 0.000,C 90.000,E1 200.120} C_DIS
LIN {X -0.036,Y -139.007,Z 1171.102,A 0.000,B 0.000,C 90.000,E1 198.290} C_DIS
LIN {X 0.051,Y -138.339,Z 1171.055,A 0.000,B 0.000,C 90.000,E1 189.849} C_DIS
LIN {X -0.065,Y -139.402,Z 1171.008,A 0.000,B 0.000,C 90.000,E1 181.489} C_DIS
LIN {X -0.012,Y -141.308,Z 1170.972,A 0.000,B 0.000,C 90.000,E1 174.951} C_DIS
LIN {X -0.055,Y -142.669,Z 1170.956,A 0.000,B 0.000,C 90.000,E1 172.186} C_DIS
LIN {X 0.067,Y -145.019,Z 1170.931,A 0.000,B 0.000,C 90.000,E1 167.521} C_DIS
LIN {X 0.025,Y -147.645,Z 1170.910,A 0.000,B 0.000,C 90.000,E1 163.866} C_DIS
LIN {X -0.040,Y -150.280,Z 1170.890,A 0.000,B 0.000,C 90.000,E1 160.242} C_DIS
LIN {X -0.027,Y -153.683,Z 1170.870,A 0.000,B 0.000,C 90.000,E1 156.613} C_DIS
LIN {X 0.028,Y -157.097,Z 1170.850,A 0.000,B 0.000,C 90.000,E1 152.999} C_DIS
LIN {X -0.033,Y -161.236,Z 1170.830,A 0.000,B 0.000,C 90.000,E1 149.459} C_DIS
LIN {X 0.052,Y -163.323,Z 1170.820,A 0.000,B 0.000,C 90.000,E1 147.661} C_DIS
LIN {X -0.077,Y -167.776,Z 1170.801,A 0.000,B 0.000,C 90.000,E1 144.196} C_DIS
LIN {X 0.075,Y -171.591,Z 1170.786,A 0.000,B 0.000,C 90.000,E1 141.537} C_DIS
LIN {X 0.005,Y -176.542,Z 1170.767,A 0.000,B 0.000,C 90.000,E1 138.119} C_DIS
LIN {X -0.002,Y -180.841,Z 1170.753,A 0.000,B 0.000,C 90.000,E1 135.567} C_DIS
LIN {X -0.018,Y -186.251,Z 1170.734,A 0.000,B 0.000,C 90.000,E1 132.204} C_DIS
LIN {X -0.080,Y -190.888,Z 1170.721,A 0.000,B 0.000,C 90.000,E1 129.725} C_DIS
LIN {X -0.048,Y -196.652,Z 1170.702,A 0.000,B 0.000,C 90.000,E1 126.423} C_DIS
LIN {X 0.114,Y -201.102,Z 1170.690,A 0.000,B 0.000,C 90.000,E1 124.119} C_DIS
LIN {X 0.141,Y -310.674,Z 1170.690,A 0.000,B 0.000,C 90.000,E1 124.119} C_DIS
LIN {X -0.128,Y -315.930,Z 1170.689,A 0.000,B 0.000,C 90.000,E1 123.992} C_DIS
LIN {X -0.154,Y -318.773,Z 1170.688,A 0.000,B 0.000,C 90.000,E1 123.785} C_DIS
LIN {X 0.145,Y -322.523,Z 1170.685,A 0.000,B 0.000,C 90.000,E1 123.293} C_DIS
LIN {X -0.010,Y -324.382,Z 1170.683,A 0.000,B 0.000,C 90.000,E1 123.007} C_DIS
LIN {X 0.106,Y -325.830,Z 1170.682,A 0.000,B 0.000,C 90.000,E1 122.673} C_DIS
LIN {X 0.062,Y -337.833,Z 1170.664,A 0.000,B 0.000,C 90.000,E1 119.539} C_DIS
LIN {X -0.109,Y -350.034,Z 1170.649,A 0.000,B 0.000,C 90.000,E1 116.796} C_DIS
LIN {X -0.102,Y -363.722,Z 1170.634,A 0.000,B 0.000,C 90.000,E1 114.079} C_DIS
LIN {X -0.098,Y -377.229,Z 1170.621,A 0.000,B 0.000,C 90.000,E1 111.716} C_DIS
LIN {X -0.027,Y -392.096,Z 1170.608,A 0.000,B 0.000,C 90.000,E1 109.396} C_DIS
LIN {X -0.094,Y -408.429,Z 1170.595,A 0.000,B 0.000,C 90.000,E1 107.149} C_DIS
LIN {X -0.125,Y -426.344,Z 1170.583,A 0.000,B 0.000,C 90.000,E1 104.954} C_DIS
LIN {X -0.137,Y -445.841,Z 1170.571,A 0.000,B 0.000,C 90.000,E1 102.827} C_DIS
LIN {X 0.024,Y -466.091,Z 1170.560,A 0.000,B 0.000,C 90.000,E1 100.838} C_DIS
LIN {X 0.067,Y -470.996,Z 1170.558,A 0.000,B 0.000,C 90.000,E1 100.366} C_DIS
LIN {X -0.105,Y -472.854,Z 1170.556,A 0.000,B 0.000,C 90.000,E1 100.141} C_DIS
LIN {X -0.193,Y -474.259,Z 1170.555,A 0.000,B 0.000,C 90.000,E1 99.905} C_DIS
LIN {X -0.002,Y -476.105,Z 1170.552,A 0.000,B 0.000,C 90.000,E1 99.378} C_DIS
LIN {X 0.121,Y -476.851,Z 1170.549,A 0.000,B 0.000,C 90.000,E1 98.859} C_DIS
LIN {X -0.214,Y -476.623,Z 1170.547,A 0.000,B 0.000,C 90.000,E1 98.398} C_DIS
LIN {X -0.005,Y -475.392,Z 1170.544,A 0.000,B 0.000,C 90.000,E1 97.871} C_DIS
LIN {X -0.203,Y -474.342,Z 1170.542,A 0.000,B 0.000,C 90.000,E1 97.644} C_DIS
LIN {X 0.133,Y -472.933,Z 1170.541,A 0.000,B 0.000,C 90.000,E1 97.352} C_DIS
LIN {X -0.176,Y -456.685,Z 1170.528,A 0.000,B 0.000,C 90.000,E1 95.106} C_DIS
LIN {X -0.019,Y -440.933,Z 1170.515,A 0.000,B 0.000,C 90.000,E1 92.751} C_DIS
LIN {X 0.082,Y -421.567,Z 1170.498,A 0.000,B 0.000,C 90.000,E1 89.542} C_DIS
LIN {X 0.138,Y -408.240,Z 1170.484,A 0.000,B 0.000,C 90.000,E1 87.078} C_DIS
LIN {X -0.180,Y -397.914,Z 1170.473,A 0.000,B 0.000,C 90.000,E1 85.179} C_DIS
LIN {X 0.114,Y -384.625,Z 1170.459,A 0.000,B 0.000,C 90.000,E1 82.591} C_DIS
LIN {X -0.154,Y -375.757,Z 1170.449,A 0.000,B 0.000,C 90.000,E1 80.905} C_DIS
LIN {X 0.162,Y -366.591,Z 1170.440,A 0.000,B 0.000,C 90.000,E1 79.106} C_DIS
LIN {X 0.008,Y -357.133,Z 1170.430,A 0.000,B 0.000,C 90.000,E1 77.353} C_DIS
LIN {X 0.188,Y -347.417,Z 1170.420,A 0.000,B 0.000,C 90.000,E1 75.519} C_DIS
LIN {X 0.069,Y -334.515,Z 1170.406,A 0.000,B 0.000,C 90.000,E1 73.087} C_DIS
LIN {X -0.063,Y -321.905,Z 1170.392,A 0.000,B 0.000,C 90.000,E1 70.604} C_DIS
LIN {X 0.055,Y -305.580,Z 1170.373,A 0.000,B 0.000,C 90.000,E1 67.050} C_DIS
LIN {X -0.045,Y -291.705,Z 1170.354,A 0.000,B 0.000,C 90.000,E1 63.768} C_DIS
LIN {X 0.000,Y -279.882,Z 1170.337,A 0.000,B 0.000,C 90.000,E1 60.717} C_DIS
LIN {X 0.054,Y -269.948,Z 1170.322,A 0.000,B 0.000,C 90.000,E1 57.946} C_DIS
LIN {X 0.145,Y -258.036,Z 1170.302,A 0.000,B 0.000,C 90.000,E1 54.402} C_DIS
LIN {X 0.108,Y -247.984,Z 1170.284,A 0.000,B 0.000,C 90.000,E1 51.170} C_DIS
LIN {X -0.109,Y -237.643,Z 1170.264,A 0.000,B 0.000,C 90.000,E1 47.553} C_DIS
LIN {X -0.005,Y -228.105,Z 1170.243,A 0.000,B 0.000,C 90.000,E1 43.785} C_DIS
LIN {X 0.000,Y -219.427,Z 1170.222,A 0.000,B 0.000,C 90.000,E1 39.967} C_DIS
LIN {X -0.032,Y -211.500,Z 1170.200,A 0.000,B 0.000,C 90.000,E1 36.091} C_DIS
LIN {X -0.004,Y -204.282,Z 1170.178,A 0.000,B 0.000,C 90.000,E1 32.133} C_DIS
LIN {X 0.060,Y -197.743,Z 1170.156,A 0.000,B 0.000,C 90.000,E1 28.103} C_DIS
LIN {X -0.091,Y -192.042,Z 1170.134,A 0.000,B 0.000,C 90.000,E1 24.079} C_DIS
LIN {X -0.020,Y -187.251,Z 1170.111,A 0.000,B 0.000,C 90.000,E1 19.939} C_DIS
LIN {X -0.054,Y -183.414,Z 1170.088,A 0.000,B 0.000,C 90.000,E1 15.788} C_DIS
LIN {X 0.055,Y -180.117,Z 1170.060,A 0.000,B 0.000,C 90.000,E1 10.715} C_DIS
LIN {X -0.031,Y -178.113,Z 1170.027,A 0.000,B 0.000,C 90.000,E1 4.821} C_DIS
LIN {X 0.038,Y -179.552,Z 1169.969,A 0.000,B 0.000,C 90.000,E1 354.432} C_DIS
LIN {X -0.063,Y -182.493,Z 1169.941,A 0.000,B 0.000,C 90.000,E1 349.398} C_DIS
LIN {X 0.043,Y -185.966,Z 1169.918,A 0.000,B 0.000,C 90.000,E1 345.172} C_DIS
LIN {X -0.043,Y -190.404,Z 1169.895,A 0.000,B 0.000,C 90.000,E1 341.040} C_DIS
LIN {X -0.035,Y -195.561,Z 1169.872,A 0.000,B 0.000,C 90.000,E1 336.922} C_DIS
LIN {X -0.094,Y -201.464,Z 1169.849,A 0.000,B 0.000,C 90.000,E1 332.871} C_DIS
LIN {X 0.040,Y -208.054,Z 1169.827,A 0.000,B 0.000,C 90.000,E1 328.820} C_DIS
LIN {X -0.072,Y -215.283,Z 1169.805,A 0.000,B 0.000,C 90.000,E1 324.895} C_DIS
LIN {X 0.053,Y -221.744,Z 1169.788,A 0.000,B 0.000,C 90.000,E1 321.743} C_DIS
LIN {X -0.040,Y -229.242,Z 1169.770,A 0.000,B 0.000,C 90.000,E1 318.690} C_DIS
LIN {X 0.001,Y -238.855,Z 1169.752,A 0.000,B 0.000,C 90.000,E1 315.283} C_DIS
LIN {X -0.006,Y -248.554,Z 1169.735,A 0.000,B 0.000,C 90.000,E1 312.324} C_DIS
LIN {X -0.049,Y -260.811,Z 1169.717,A 0.000,B 0.000,C 90.000,E1 309.072} C_DIS
LIN {X -0.019,Y -271.183,Z 1169.703,A 0.000,B 0.000,C 90.000,E1 306.583} C_DIS
LIN {X 0.137,Y -282.656,Z 1169.690,A 0.000,B 0.000,C 90.000,E1 304.119} C_DIS
LIN {X 0.085,Y -297.398,Z 1169.675,A 0.000,B 0.000,C 90.000,E1 301.416} C_DIS
LIN {X -0.086,Y -309.358,Z 1169.664,A 0.000,B 0.000,C 90.000,E1 299.461} C_DIS
LIN {X -0.139,Y -320.066,Z 1169.655,A 0.000,B 0.000,C 90.000,E1 297.847} C_DIS
LIN {X -0.024,Y -331.857,Z 1169.646,A 0.000,B 0.000,C 90.000,E1 296.232} C_DIS
LIN {X 0.004,Y -352.520,Z 1169.632,A 0.000,B 0.000,C 90.000,E1 293.770} C_DIS
LIN {X 0.077,Y -368.406,Z 1169.623,A 0.000,B 0.000,C 90.000,E1 292.078} C_DIS
LIN {X -0.083,Y -390.114,Z 1169.611,A 0.000,B 0.000,C 90.000,E1 290.066} C_DIS
LIN {X -0.171,Y -400.785,Z 1169.606,A 0.000,B 0.000,C 90.000,E1 289.087} C_DIS
LIN {X -0.036,Y -408.711,Z 1169.602,A 0.000,B 0.000,C 90.000,E1 288.308} C_DIS
LIN {X 0.007,Y -418.904,Z 1169.596,A 0.000,B 0.000,C 90.000,E1 287.275} C_DIS
LIN {X -0.030,Y -426.361,Z 1169.592,A 0.000,B 0.000,C 90.000,E1 286.496} C_DIS
LIN {X 0.198,Y -433.582,Z 1169.587,A 0.000,B 0.000,C 90.000,E1 285.662} C_DIS
LIN {X -0.088,Y -440.312,Z 1169.583,A 0.000,B 0.000,C 90.000,E1 284.898} C_DIS
LIN {X -0.201,Y -446.232,Z 1169.578,A 0.000,B 0.000,C 90.000,E1 284.120} C_DIS
LIN {X 0.059,Y -451.486,Z 1169.574,A 0.000,B 0.000,C 90.000,E1 283.300} C_DIS
LIN {X -0.064,Y -456.102,Z 1169.570,A 0.000,B 0.000,C 90.000,E1 282.535} C_DIS
LIN {X -0.154,Y -460.097,Z 1169.565,A 0.000,B 0.000,C 90.000,E1 281.771} C_DIS
LIN {X 0.246,Y -463.454,Z 1169.561,A 0.000,B 0.000,C 90.000,E1 280.950} C_DIS
LIN {X 0.134,Y -466.367,Z 1169.557,A 0.000,B 0.000,C 90.000,E1 280.197} C_DIS
LIN {X -0.184,Y -468.074,Z 1169.554,A 0.000,B 0.000,C 90.000,E1 279.726} C_DIS
LIN {X -0.110,Y -469.586,Z 1169.551,A 0.000,B 0.000,C 90.000,E1 279.208} C_DIS
LIN {X 0.049,Y -470.821,Z 1169.548,A 0.000,B 0.000,C 90.000,E1 278.681} C_DIS
LIN {X 0.145,Y -471.776,Z 1169.545,A 0.000,B 0.000,C 90.000,E1 278.163} C_DIS
LIN {X -0.217,Y -472.439,Z 1169.543,A 0.000,B 0.000,C 90.000,E1 277.701} C_DIS
LIN {X -0.104,Y -472.749,Z 1169.540,A 0.000,B 0.000,C 90.000,E1 277.182} C_DIS
LIN {X 0.014,Y -472.652,Z 1169.537,A 0.000,B 0.000,C 90.000,E1 276.663} C_DIS
LIN {X 0.133,Y -472.147,Z 1169.534,A 0.000,B 0.000,C 90.000,E1 276.144} C_DIS
LIN {X -0.218,Y -471.217,Z 1169.531,A 0.000,B 0.000,C 90.000,E1 275.682} C_DIS
LIN {X -0.102,Y -469.809,Z 1169.529,A 0.000,B 0.000,C 90.000,E1 275.163} C_DIS
LIN {X 0.005,Y -467.950,Z 1169.526,A 0.000,B 0.000,C 90.000,E1 274.645} C_DIS
LIN {X 0.068,Y -465.536,Z 1169.523,A 0.000,B 0.000,C 90.000,E1 274.131} C_DIS
LIN {X 0.147,Y -462.469,Z 1169.520,A 0.000,B 0.000,C 90.000,E1 273.612} C_DIS
LIN {X -0.066,Y -460.661,Z 1169.519,A 0.000,B 0.000,C 90.000,E1 273.383} C_DIS
LIN {X -0.016,Y -456.274,Z 1169.516,A 0.000,B 0.000,C 90.000,E1 272.865} C_DIS
LIN {X 0.219,Y -453.691,Z 1169.515,A 0.000,B 0.000,C 90.000,E1 272.579} C_DIS
LIN {X -0.103,Y -447.597,Z 1169.512,A 0.000,B 0.000,C 90.000,E1 272.121} C_DIS
LIN {X 0.028,Y -444.507,Z 1169.510,A 0.000,B 0.000,C 90.000,E1 271.892} C_DIS
LIN {X 0.145,Y -437.814,Z 1169.508,A 0.000,B 0.000,C 90.000,E1 271.489} C_DIS
LIN {X -0.095,Y -430.829,Z 1169.507,A 0.000,B 0.000,C 90.000,E1 271.203} C_DIS
LIN {X 0.077,Y -423.931,Z 1169.505,A 0.000,B 0.000,C 90.000,E1 270.917} C_DIS
LIN {X 0.120,Y -416.993,Z 1169.504,A 0.000,B 0.000,C 90.000,E1 270.688} C_DIS
LIN {X 0.006,Y -409.775,Z 1169.503,A 0.000,B 0.000,C 90.000,E1 270.516} C_DIS
LIN {X 0.015,Y -399.124,Z 1169.502,A 0.000,B 0.000,C 90.000,E1 270.286} C_DIS
LIN {X -0.083,Y -388.552,Z 1169.501,A 0.000,B 0.000,C 90.000,E1 270.115} C_DIS
LIN {X -0.033,Y -379.713,Z 1169.500,A 0.000,B 0.000,C 90.000,E1 270.000} C_DIS
LIN {X -0.030,Y -371.251,Z 1169.500,A 0.000,B 0.000,C 90.000,E1 269.943} C_DIS
LIN {X -0.042,Y -181.548,Z 1169.500,A 0.000,B 0.000,C 90.000,E1 269.943} C_DIS
LIN {X -0.042,Y -180.812,Z 1169.471,A 0.000,B 0.000,C 90.000,E1 264.837} C_DIS
LIN {X 0.035,Y -178.915,Z 1169.443,A 0.000,B 0.000,C 90.000,E1 259.746} C_DIS
LIN {X -0.055,Y -175.960,Z 1169.415,A 0.000,B 0.000,C 90.000,E1 254.685} C_DIS
LIN {X 0.061,Y -175.433,Z 1169.410,A 0.000,B 0.000,C 90.000,E1 253.795} C_DIS
LIN {X 0.064,Y -172.192,Z 1169.386,A 0.000,B 0.000,C 90.000,E1 249.518} C_DIS
LIN {X 0.040,Y -171.664,Z 1169.382,A 0.000,B 0.000,C 90.000,E1 248.666} C_DIS
LIN {X 0.024,Y -167.890,Z 1169.358,A 0.000,B 0.000,C 90.000,E1 244.357} C_DIS
LIN {X 0.039,Y -166.627,Z 1169.348,A 0.000,B 0.000,C 90.000,E1 242.615} C_DIS
LIN {X 0.032,Y -162.613,Z 1169.324,A 0.000,B 0.000,C 90.000,E1 238.250} C_DIS
LIN {X 0.005,Y -161.299,Z 1169.314,A 0.000,B 0.000,C 90.000,E1 236.501} C_DIS
LIN {X 0.040,Y -157.297,Z 1169.289,A 0.000,B 0.000,C 90.000,E1 232.065} C_DIS
LIN {X 0.069,Y -155.272,Z 1169.274,A 0.000,B 0.000,C 90.000,E1 229.380} C_DIS
LIN {X -0.003,Y -151.639,Z 1169.250,A 0.000,B 0.000,C 90.000,E1 224.919} C_DIS
LIN {X 0.045,Y -150.508,Z 1169.240,A 0.000,B 0.000,C 90.000,E1 223.095} C_DIS
LIN {X 0.073,Y -147.232,Z 1169.214,A 0.000,B 0.000,C 90.000,E1 218.543} C_DIS
LIN {X 0.043,Y -145.256,Z 1169.194,A 0.000,B 0.000,C 90.000,E1 214.898} C_DIS
LIN {X -0.041,Y -142.369,Z 1169.163,A 0.000,B 0.000,C 90.000,E1 209.411} C_DIS
LIN {X 0.079,Y -141.754,Z 1169.153,A 0.000,B 0.000,C 90.000,E1 207.513} C_DIS
LIN {X 0.005,Y -139.496,Z 1169.117,A 0.000,B 0.000,C 90.000,E1 201.046} C_DIS
LIN {X 0.042,Y -139.001,Z 1169.101,A 0.000,B 0.000,C 90.000,E1 198.236} C_DIS
LIN {X -0.001,Y -138.338,Z 1169.055,A 0.000,B 0.000,C 90.000,E1 189.849} C_DIS
LIN {X 0.021,Y -139.409,Z 1169.008,A 0.000,B 0.000,C 90.000,E1 181.432} C_DIS
LIN {X -0.067,Y -141.319,Z 1168.972,A 0.000,B 0.000,C 90.000,E1 174.951} C_DIS
LIN {X 0.032,Y -142.678,Z 1168.956,A 0.000,B 0.000,C 90.000,E1 172.129} C_DIS
LIN {X 0.012,Y -145.033,Z 1168.931,A 0.000,B 0.000,C 90.000,E1 167.521} C_DIS
LIN {X -0.031,Y -147.658,Z 1168.910,A 0.000,B 0.000,C 90.000,E1 163.866} C_DIS
LIN {X 0.045,Y -150.297,Z 1168.890,A 0.000,B 0.000,C 90.000,E1 160.188} C_DIS
LIN {X -0.084,Y -153.706,Z 1168.870,A 0.000,B 0.000,C 90.000,E1 156.613} C_DIS
LIN {X -0.029,Y -157.119,Z 1168.850,A 0.000,B 0.000,C 90.000,E1 152.999} C_DIS
LIN {X 0.047,Y -161.263,Z 1168.830,A 0.000,B 0.000,C 90.000,E1 149.410} C_DIS
LIN {X -0.026,Y -164.381,Z 1168.815,A 0.000,B 0.000,C 90.000,E1 146.786} C_DIS
LIN {X -0.039,Y -169.056,Z 1168.796,A 0.000,B 0.000,C 90.000,E1 143.290} C_DIS
LIN {X 0.014,Y -171.618,Z 1168.786,A 0.000,B 0.000,C 90.000,E1 141.537} C_DIS
LIN {X 0.061,Y -176.574,Z 1168.767,A 0.000,B 0.000,C 90.000,E1 138.081} C_DIS
LIN {X -0.065,Y -180.872,Z 1168.753,A 0.000,B 0.000,C 90.000,E1 135.567} C_DIS
LIN {X 0.056,Y -186.286,Z 1168.734,A 0.000,B 0.000,C 90.000,E1 132.162} C_DIS
LIN {X -0.023,Y -190.921,Z 1168.720,A 0.000,B 0.000,C 90.000,E1 129.688} C_DIS
LIN {X 0.044,Y -196.689,Z 1168.702,A 0.000,B 0.000,C 90.000,E1 126.377} C_DIS
LIN {X -0.113,Y -201.076,Z 1168.690,A 0.000,B 0.000,C 90.000,E1 124.199} C_DIS
LIN {X -0.211,Y -310.294,Z 1168.690,A 0.000,B 0.000,C 90.000,E1 124.199} C_DIS
LIN {X 0.206,Y -316.367,Z 1168.689,A 0.000,B 0.000,C 90.000,E1 123.913} C_DIS
LIN {X 0.036,Y -319.312,Z 1168.687,A 0.000,B 0.000,C 90.000,E1 123.706} C_DIS
LIN {X -0.018,Y -323.036,Z 1168.685,A 0.000,B 0.000,C 90.000,E1 123.245} C_DIS
LIN {X 0.063,Y -324.795,Z 1168.683,A 0.000,B 0.000,C 90.000,E1 122.911} C_DIS
LIN {X -0.032,Y -327.302,Z 1168.679,A 0.000,B 0.000,C 90.000,E1 122.291} C_DIS
LIN {X 0.004,Y -338.173,Z 1168.664,A 0.000,B 0.000,C 90.000,E1 119.461} C_DIS
LIN {X -0.012,Y -350.420,Z 1168.648,A 0.000,B 0.000,C 90.000,E1 116.693} C_DIS
LIN {X 0.174,Y -364.156,Z 1168.633,A 0.000,B 0.000,C 90.000,E1 113.951} C_DIS
LIN {X 0.198,Y -377.708,Z 1168.620,A 0.000,B 0.000,C 90.000,E1 111.589} C_DIS
LIN {X -0.081,Y -392.625,Z 1168.607,A 0.000,B 0.000,C 90.000,E1 109.322} C_DIS
LIN {X 0.123,Y -409.013,Z 1168.595,A 0.000,B 0.000,C 90.000,E1 107.040} C_DIS
LIN {X 0.234,Y -426.985,Z 1168.583,A 0.000,B 0.000,C 90.000,E1 104.828} C_DIS
LIN {X 0.165,Y -446.524,Z 1168.571,A 0.000,B 0.000,C 90.000,E1 102.715} C_DIS
LIN {X -0.065,Y -466.794,Z 1168.560,A 0.000,B 0.000,C 90.000,E1 100.782} C_DIS
LIN {X -0.038,Y -469.349,Z 1168.559,A 0.000,B 0.000,C 90.000,E1 100.546} C_DIS
LIN {X -0.011,Y -471.502,Z 1168.557,A 0.000,B 0.000,C 90.000,E1 100.310} C_DIS
LIN {X -0.158,Y -473.258,Z 1168.556,A 0.000,B 0.000,C 90.000,E1 100.074} C_DIS
LIN {X 0.080,Y -474.577,Z 1168.554,A 0.000,B 0.000,C 90.000,E1 99.792} C_DIS
LIN {X -0.194,Y -476.219,Z 1168.552,A 0.000,B 0.000,C 90.000,E1 99.321} C_DIS
LIN {X -0.069,Y -476.799,Z 1168.549,A 0.000,B 0.000,C 90.000,E1 98.803} C_DIS
LIN {X 0.138,Y -476.409,Z 1168.546,A 0.000,B 0.000,C 90.000,E1 98.276} C_DIS
LIN {X -0.194,Y -474.996,Z 1168.543,A 0.000,B 0.000,C 90.000,E1 97.814} C_DIS
LIN {X 0.080,Y -473.835,Z 1168.542,A 0.000,B 0.000,C 90.000,E1 97.530} C_DIS
LIN {X -0.055,Y -472.286,Z 1168.541,A 0.000,B 0.000,C 90.000,E1 97.296} C_DIS
LIN {X 0.083,Y -455.998,Z 1168.528,A 0.000,B 0.000,C 90.000,E1 94.992} C_DIS
LIN {X 0.217,Y -440.313,Z 1168.515,A 0.000,B 0.000,C 90.000,E1 92.636} C_DIS
LIN {X 0.165,Y -422.525,Z 1168.499,A 0.000,B 0.000,C 90.000,E1 89.714} C_DIS
LIN {X -0.159,Y -409.172,Z 1168.485,A 0.000,B 0.000,C 90.000,E1 87.306} C_DIS
LIN {X -0.089,Y -398.845,Z 1168.474,A 0.000,B 0.000,C 90.000,E1 85.355} C_DIS
LIN {X -0.113,Y -385.527,Z 1168.460,A 0.000,B 0.000,C 90.000,E1 82.818} C_DIS
LIN {X -0.041,Y -376.678,Z 1168.450,A 0.000,B 0.000,C 90.000,E1 81.084} C_DIS
LIN {X -0.077,Y -367.530,Z 1168.441,A 0.000,B 0.000,C 90.000,E1 79.342} C_DIS
LIN {X -0.210,Y -358.098,Z 1168.431,A 0.000,B 0.000,C 90.000,E1 77.589} C_DIS
LIN {X -0.006,Y -348.397,Z 1168.421,A 0.000,B 0.000,C 90.000,E1 75.755} C_DIS
LIN {X 0.009,Y -337.070,Z 1168.409,A 0.000,B 0.000,C 90.000,E1 73.614} C_DIS
LIN {X 0.152,Y -324.355,Z 1168.395,A 0.000,B 0.000,C 90.000,E1 71.094} C_DIS
LIN {X -0.062,Y -307.843,Z 1168.376,A 0.000,B 0.000,C 90.000,E1 67.614} C_DIS
LIN {X -0.090,Y -293.845,Z 1168.357,A 0.000,B 0.000,C 90.000,E1 64.332} C_DIS
LIN {X -0.112,Y -281.904,Z 1168.340,A 0.000,B 0.000,C 90.000,E1 61.307} C_DIS
LIN {X -0.062,Y -270.609,Z 1168.323,A 0.000,B 0.000,C 90.000,E1 58.201} C_DIS
LIN {X -0.087,Y -258.625,Z 1168.304,A 0.000,B 0.000,C 90.000,E1 54.689} C_DIS
LIN {X -0.102,Y -248.522,Z 1168.286,A 0.000,B 0.000,C 90.000,E1 51.457} C_DIS
LIN {X -0.102,Y -239.113,Z 1168.267,A 0.000,B 0.000,C 90.000,E1 48.162} C_DIS
LIN {X -0.110,Y -229.458,Z 1168.247,A 0.000,B 0.000,C 90.000,E1 44.433} C_DIS
LIN {X -0.079,Y -220.635,Z 1168.226,A 0.000,B 0.000,C 90.000,E1 40.620} C_DIS
LIN {X 0.054,Y -212.546,Z 1168.204,A 0.000,B 0.000,C 90.000,E1 36.710} C_DIS
LIN {X 0.108,Y -205.219,Z 1168.182,A 0.000,B 0.000,C 90.000,E1 32.752} C_DIS
LIN {X 0.029,Y -198.500,Z 1168.160,A 0.000,B 0.000,C 90.000,E1 28.771} C_DIS
LIN {X -0.007,Y -192.626,Z 1168.137,A 0.000,B 0.000,C 90.000,E1 24.719} C_DIS
LIN {X -0.021,Y -187.677,Z 1168.115,A 0.000,B 0.000,C 90.000,E1 20.610} C_DIS
LIN {X 0.013,Y -183.679,Z 1168.091,A 0.000,B 0.000,C 90.000,E1 16.441} C_DIS
LIN {X -0.043,Y -180.171,Z 1168.063,A 0.000,B 0.000,C 90.000,E1 11.422} C_DIS
LIN {X -0.017,Y -177.793,Z 1168.026,A 0.000,B 0.000,C 90.000,E1 4.645} C_DIS
LIN {X 0.026,Y -179.209,Z 1167.969,A 0.000,B 0.000,C 90.000,E1 354.432} C_DIS
LIN {X -0.087,Y -182.150,Z 1167.941,A 0.000,B 0.000,C 90.000,E1 349.398} C_DIS
LIN {X 0.007,Y -185.630,Z 1167.918,A 0.000,B 0.000,C 90.000,E1 345.172} C_DIS
LIN {X -0.090,Y -190.039,Z 1167.895,A 0.000,B 0.000,C 90.000,E1 341.040} C_DIS
LIN {X -0.096,Y -195.197,Z 1167.872,A 0.000,B 0.000,C 90.000,E1 336.922} C_DIS
LIN {X 0.011,Y -201.076,Z 1167.849,A 0.000,B 0.000,C 90.000,E1 332.820} C_DIS
LIN {X 0.059,Y -207.677,Z 1167.827,A 0.000,B 0.000,C 90.000,E1 328.791} C_DIS
LIN {X 0.001,Y -214.959,Z 1167.805,A 0.000,B 0.000,C 90.000,E1 324.848} C_DIS
LIN {X -0.062,Y -221.456,Z 1167.787,A 0.000,B 0.000,C 90.000,E1 321.743} C_DIS
LIN {X 0.071,Y -227.999,Z 1167.772,A 0.000,B 0.000,C 90.000,E1 319.013} C_DIS
LIN {X -0.093,Y -237.538,Z 1167.753,A 0.000,B 0.000,C 90.000,E1 315.648} C_DIS
LIN {X -0.144,Y -247.136,Z 1167.737,A 0.000,B 0.000,C 90.000,E1 312.690} C_DIS
LIN {X 0.093,Y -257.896,Z 1167.721,A 0.000,B 0.000,C 90.000,E1 309.725} C_DIS
LIN {X 0.127,Y -269.611,Z 1167.705,A 0.000,B 0.000,C 90.000,E1 306.870} C_DIS
LIN {X -0.029,Y -282.685,Z 1167.690,A 0.000,B 0.000,C 90.000,E1 304.119} C_DIS
LIN {X 0.068,Y -299.383,Z 1167.673,A 0.000,B 0.000,C 90.000,E1 301.052} C_DIS
LIN {X 0.045,Y -311.554,Z 1167.662,A 0.000,B 0.000,C 90.000,E1 299.077} C_DIS
LIN {X 0.027,Y -322.463,Z 1167.653,A 0.000,B 0.000,C 90.000,E1 297.462} C_DIS
LIN {X -0.144,Y -336.987,Z 1167.642,A 0.000,B 0.000,C 90.000,E1 295.591} C_DIS
LIN {X -0.180,Y -357.737,Z 1167.629,A 0.000,B 0.000,C 90.000,E1 293.206} C_DIS
LIN {X -0.035,Y -370.796,Z 1167.621,A 0.000,B 0.000,C 90.000,E1 291.844} C_DIS
LIN {X 0.143,Y -389.623,Z 1167.612,A 0.000,B 0.000,C 90.000,E1 290.066} C_DIS
LIN {X 0.138,Y -400.209,Z 1167.606,A 0.000,B 0.000,C 90.000,E1 289.087} C_DIS
LIN {X -0.128,Y -410.768,Z 1167.600,A 0.000,B 0.000,C 90.000,E1 288.109} C_DIS
LIN {X 0.091,Y -421.011,Z 1167.595,A 0.000,B 0.000,C 90.000,E1 287.040} C_DIS
LIN {X 0.007,Y -428.430,Z 1167.590,A 0.000,B 0.000,C 90.000,E1 286.260} C_DIS
LIN {X -0.154,Y -435.497,Z 1167.586,A 0.000,B 0.000,C 90.000,E1 285.481} C_DIS
LIN {X 0.004,Y -442.033,Z 1167.581,A 0.000,B 0.000,C 90.000,E1 284.662} C_DIS
LIN {X -0.100,Y -447.776,Z 1167.577,A 0.000,B 0.000,C 90.000,E1 283.883} C_DIS
LIN {X 0.182,Y -452.848,Z 1167.573,A 0.000,B 0.000,C 90.000,E1 283.063} C_DIS
LIN {X 0.067,Y -457.306,Z 1167.568,A 0.000,B 0.000,C 90.000,E1 282.299} C_DIS
LIN {X -0.008,Y -461.120,Z 1167.564,A 0.000,B 0.000,C 90.000,E1 281.535} C_DIS
LIN {X -0.145,Y -464.387,Z 1167.560,A 0.000,B 0.000,C 90.000,E1 280.782} C_DIS
LIN {X 0.135,Y -468.045,Z 1167.554,A 0.000,B 0.000,C 90.000,E1 279.726} C_DIS
LIN {X 0.209,Y -469.587,Z 1167.551,A 0.000,B 0.000,C 90.000,E1 279.208} C_DIS
LIN {X -0.167,Y -470.849,Z 1167.548,A 0.000,B 0.000,C 90.000,E1 278.746} C_DIS
LIN {X 0.000,Y -471.858,Z 1167.546,A 0.000,B 0.000,C 90.000,E1 278.219} C_DIS
LIN {X 0.105,Y -472.587,Z 1167.543,A 0.000,B 0.000,C 90.000,E1 277.701} C_DIS
LIN {X 0.219,Y -472.942,Z 1167.540,A 0.000,B 0.000,C 90.000,E1 277.182} C_DIS
LIN {X -0.132,Y -472.905,Z 1167.537,A 0.000,B 0.000,C 90.000,E1 276.720} C_DIS
LIN {X -0.012,Y -472.441,Z 1167.534,A 0.000,B 0.000,C 90.000,E1 276.201} C_DIS
LIN {X 0.108,Y -471.578,Z 1167.532,A 0.000,B 0.000,C 90.000,E1 275.682} C_DIS
LIN {X 0.223,Y -470.265,Z 1167.529,A 0.000,B 0.000,C 90.000,E1 275.163} C_DIS
LIN {X -0.135,Y -468.445,Z 1167.526,A 0.000,B 0.000,C 90.000,E1 274.702} C_DIS
LIN {X -0.069,Y -466.109,Z 1167.523,A 0.000,B 0.000,C 90.000,E1 274.188} C_DIS
LIN {X 0.013,Y -463.100,Z 1167.520,A 0.000,B 0.000,C 90.000,E1 273.669} C_DIS
LIN {X -0.198,Y -461.357,Z 1167.519,A 0.000,B 0.000,C 90.000,E1 273.440} C_DIS
LIN {X -0.142,Y -457.074,Z 1167.516,A 0.000,B 0.000,C 90.000,E1 272.922} C_DIS
LIN {X 0.095,Y -454.573,Z 1167.515,A 0.000,B 0.000,C 90.000,E1 272.636} C_DIS
LIN {X -0.103,Y -451.749,Z 1167.513,A 0.000,B 0.000,C 90.000,E1 272.407} C_DIS
LIN {X 0.151,Y -448.585,Z 1167.512,A 0.000,B 0.000,C 90.000,E1 272.121} C_DIS
LIN {X -0.096,Y -441.966,Z 1167.510,A 0.000,B 0.000,C 90.000,E1 271.718} C_DIS
LIN {X -0.157,Y -438.763,Z 1167.508,A 0.000,B 0.000,C 90.000,E1 271.547} C_DIS
LIN {X -0.012,Y -431.806,Z 1167.507,A 0.000,B 0.000,C 90.000,E1 271.203} C_DIS
LIN {X 0.070,Y -421.344,Z 1167.505,A 0.000,B 0.000,C 90.000,E1 270.802} C_DIS
LIN {X 0.159,Y -413.928,Z 1167.503,A 0.000,B 0.000,C 90.000,E1 270.573} C_DIS
LIN {X 0.043,Y -403.290,Z 1167.502,A 0.000,B 0.000,C 90.000,E1 270.344} C_DIS
LIN {X -0.141,Y -389.461,Z 1167.500,A 0.000,B 0.000,C 90.000,E1 270.115} C_DIS
LIN {X -0.085,Y -380.997,Z 1167.500,A 0.000,B 0.000,C 90.000,E1 270.000} C_DIS
LIN {X -0.145,Y -369.561,Z 1167.500,A 0.000,B 0.000,C 90.000,E1 269.943} C_DIS
LIN {X 0.082,Y -181.544,Z 1167.500,A 0.000,B 0.000,C 90.000,E1 269.885} C_DIS
LIN {X -0.076,Y -180.810,Z 1167.471,A 0.000,B 0.000,C 90.000,E1 264.837} C_DIS
LIN {X 0.001,Y -178.910,Z 1167.443,A 0.000,B 0.000,C 90.000,E1 259.746} C_DIS
LIN {X 0.081,Y -175.955,Z 1167.415,A 0.000,B 0.000,C 90.000,E1 254.629} C_DIS
LIN {X 0.027,Y -175.424,Z 1167.410,A 0.000,B 0.000,C 90.000,E1 253.795} C_DIS
LIN {X 0.030,Y -172.185,Z 1167.386,A 0.000,B 0.000,C 90.000,E1 249.518} C_DIS
LIN {X 0.069,Y -171.657,Z 1167.381,A 0.000,B 0.000,C 90.000,E1 248.646} C_DIS
LIN {X 0.064,Y -167.881,Z 1167.358,A 0.000,B 0.000,C 90.000,E1 244.332} C_DIS
LIN {X 0.006,Y -166.617,Z 1167.348,A 0.000,B 0.000,C 90.000,E1 242.615} C_DIS
LIN {X 0.000,Y -162.605,Z 1167.324,A 0.000,B 0.000,C 90.000,E1 238.250} C_DIS
LIN {X -0.026,Y -161.289,Z 1167.314,A 0.000,B 0.000,C 90.000,E1 236.501} C_DIS
LIN {X 0.009,Y -157.288,Z 1167.289,A 0.000,B 0.000,C 90.000,E1 232.065} C_DIS
LIN {X 0.031,Y -156.005,Z 1167.279,A 0.000,B 0.000,C 90.000,E1 230.275} C_DIS
LIN {X -0.009,Y -152.263,Z 1167.255,A 0.000,B 0.000,C 90.000,E1 225.810} C_DIS
LIN {X 0.013,Y -150.501,Z 1167.240,A 0.000,B 0.000,C 90.000,E1 223.095} C_DIS
LIN {X 0.043,Y -147.226,Z 1167.214,A 0.000,B 0.000,C 90.000,E1 218.543} C_DIS
LIN {X 0.012,Y -145.248,Z 1167.194,A 0.000,B 0.000,C 90.000,E1 214.898} C_DIS
LIN {X -0.071,Y -142.365,Z 1167.163,A 0.000,B 0.000,C 90.000,E1 209.411} C_DIS
LIN {X 0.050,Y -141.750,Z 1167.153,A 0.000,B 0.000,C 90.000,E1 207.513} C_DIS
LIN {X -0.024,Y -139.493,Z 1167.117,A 0.000,B 0.000,C 90.000,E1 201.046} C_DIS
LIN {X 0.013,Y -138.998,Z 1167.101,A 0.000,B 0.000,C 90.000,E1 198.236} C_DIS
LIN {X -0.030,Y -138.337,Z 1167.055,A 0.000,B 0.000,C 90.000,E1 189.849} C_DIS
LIN {X -0.009,Y -139.411,Z 1167.008,A 0.000,B 0.000,C 90.000,E1 181.432} C_DIS
LIN {X 0.044,Y -141.324,Z 1166.972,A 0.000,B 0.000,C 90.000,E1 174.894} C_DIS
LIN {X 0.002,Y -142.682,Z 1166.956,A 0.000,B 0.000,C 90.000,E1 172.129} C_DIS
LIN {X -0.018,Y -145.040,Z 1166.931,A 0.000,B 0.000,C 90.000,E1 167.521} C_DIS
LIN {X -0.021,Y -147.666,Z 1166.910,A 0.000,B 0.000,C 90.000,E1 163.850} C_DIS
LIN {X 0.015,Y -150.307,Z 1166.890,A 0.000,B 0.000,C 90.000,E1 160.188} C_DIS
LIN {X 0.026,Y -153.718,Z 1166.870,A 0.000,B 0.000,C 90.000,E1 156.561} C_DIS
LIN {X -0.061,Y -157.132,Z 1166.850,A 0.000,B 0.000,C 90.000,E1 152.999} C_DIS
LIN {X 0.014,Y -161.278,Z 1166.830,A 0.000,B 0.000,C 90.000,E1 149.410} C_DIS
LIN {X 0.031,Y -164.394,Z 1166.815,A 0.000,B 0.000,C 90.000,E1 146.755} C_DIS
LIN {X 0.029,Y -169.073,Z 1166.796,A 0.000,B 0.000,C 90.000,E1 143.256} C_DIS
LIN {X -0.020,Y -171.632,Z 1166.786,A 0.000,B 0.000,C 90.000,E1 141.537} C_DIS
LIN {X 0.027,Y -176.591,Z 1166.767,A 0.000,B 0.000,C 90.000,E1 138.081} C_DIS
LIN {X -0.100,Y -180.889,Z 1166.753,A 0.000,B 0.000,C 90.000,E1 135.567} C_DIS
LIN {X 0.020,Y -186.305,Z 1166.734,A 0.000,B 0.000,C 90.000,E1 132.162} C_DIS
LIN {X 0.088,Y -190.939,Z 1166.720,A 0.000,B 0.000,C 90.000,E1 129.644} C_DIS
LIN {X 0.008,Y -196.709,Z 1166.702,A 0.000,B 0.000,C 90.000,E1 126.377} C_DIS
LIN {X -0.072,Y -201.056,Z 1166.690,A 0.000,B 0.000,C 90.000,E1 124.199} C_DIS
LIN {X -0.153,Y -310.345,Z 1166.690,A 0.000,B 0.000,C 90.000,E1 124.199} C_DIS
LIN {X 0.147,Y -316.640,Z 1166.689,A 0.000,B 0.000,C 90.000,E1 123.913} C_DIS
LIN {X 0.016,Y -319.401,Z 1166.687,A 0.000,B 0.000,C 90.000,E1 123.706} C_DIS
LIN {X 0.063,Y -323.151,Z 1166.685,A 0.000,B 0.000,C 90.000,E1 123.214} C_DIS
LIN {X 0.143,Y -324.870,Z 1166.683,A 0.000,B 0.000,C 90.000,E1 122.880} C_DIS
LIN {X 0.047,Y -327.341,Z 1166.679,A 0.000,B 0.000,C 90.000,E1 122.260} C_DIS
LIN {X -0.095,Y -338.220,Z 1166.664,A 0.000,B 0.000,C 90.000,E1 119.461} C_DIS
LIN {X 0.045,Y -350.475,Z 1166.648,A 0.000,B 0.000,C 90.000,E1 116.668} C_DIS
LIN {X 0.071,Y -364.219,Z 1166.633,A 0.000,B 0.000,C 90.000,E1 113.951} C_DIS
LIN {X 0.092,Y -377.782,Z 1166.620,A 0.000,B 0.000,C 90.000,E1 111.589} C_DIS
LIN {X 0.182,Y -392.708,Z 1166.607,A 0.000,B 0.000,C 90.000,E1 109.268} C_DIS
LIN {X 0.013,Y -409.105,Z 1166.595,A 0.000,B 0.000,C 90.000,E1 107.040} C_DIS
LIN {X 0.121,Y -427.089,Z 1166.583,A 0.000,B 0.000,C 90.000,E1 104.828} C_DIS
LIN {X 0.052,Y -446.636,Z 1166.571,A 0.000,B 0.000,C 90.000,E1 102.715} C_DIS
LIN {X -0.173,Y -466.910,Z 1166.560,A 0.000,B 0.000,C 90.000,E1 100.782} C_DIS
LIN {X -0.146,Y -469.457,Z 1166.558,A 0.000,B 0.000,C 90.000,E1 100.546} C_DIS
LIN {X -0.120,Y -471.559,Z 1166.557,A 0.000,B 0.000,C 90.000,E1 100.310} C_DIS
LIN {X 0.200,Y -473.281,Z 1166.556,A 0.000,B 0.000,C 90.000,E1 100.018} C_DIS
LIN {X -0.028,Y -474.572,Z 1166.554,A 0.000,B 0.000,C 90.000,E1 99.792} C_DIS
LIN {X 0.167,Y -476.175,Z 1166.552,A 0.000,B 0.000,C 90.000,E1 99.265} C_DIS
LIN {X -0.177,Y -476.720,Z 1166.549,A 0.000,B 0.000,C 90.000,E1 98.803} C_DIS
LIN {X 0.030,Y -476.298,Z 1166.546,A 0.000,B 0.000,C 90.000,E1 98.276} C_DIS
LIN {X 0.169,Y -474.847,Z 1166.543,A 0.000,B 0.000,C 90.000,E1 97.757} C_DIS
LIN {X -0.029,Y -473.662,Z 1166.542,A 0.000,B 0.000,C 90.000,E1 97.530} C_DIS
LIN {X -0.163,Y -472.083,Z 1166.540,A 0.000,B 0.000,C 90.000,E1 97.296} C_DIS
LIN {X -0.027,Y -455.809,Z 1166.528,A 0.000,B 0.000,C 90.000,E1 94.992} C_DIS
LIN {X 0.106,Y -440.134,Z 1166.515,A 0.000,B 0.000,C 90.000,E1 92.636} C_DIS
LIN {X 0.176,Y -420.835,Z 1166.497,A 0.000,B 0.000,C 90.000,E1 89.427} C_DIS
LIN {X 0.138,Y -409.030,Z 1166.485,A 0.000,B 0.000,C 90.000,E1 87.249} C_DIS
LIN {X -0.201,Y -398.692,Z 1166.474,A 0.000,B 0.000,C 90.000,E1 85.355} C_DIS
LIN {X 0.157,Y -385.357,Z 1166.460,A 0.000,B 0.000,C 90.000,E1 82.761} C_DIS
LIN {X -0.154,Y -376.486,Z 1166.450,A 0.000,B 0.000,C 90.000,E1 81.084} C_DIS
LIN {X -0.190,Y -367.333,Z 1166.441,A 0.000,B 0.000,C 90.000,E1 79.342} C_DIS
LIN {X 0.102,Y -357.879,Z 1166.431,A 0.000,B 0.000,C 90.000,E1 77.521} C_DIS
LIN {X -0.122,Y -348.183,Z 1166.421,A 0.000,B 0.000,C 90.000,E1 75.755} C_DIS
LIN {X -0.108,Y -336.843,Z 1166.409,A 0.000,B 0.000,C 90.000,E1 73.614} C_DIS
LIN {X 0.034,Y -324.118,Z 1166.395,A 0.000,B 0.000,C 90.000,E1 71.094} C_DIS
LIN {X -0.064,Y -307.619,Z 1166.375,A 0.000,B 0.000,C 90.000,E1 67.592} C_DIS
LIN {X 0.054,Y -295.009,Z 1166.359,A 0.000,B 0.000,C 90.000,E1 64.613} C_DIS
LIN {X 0.048,Y -282.993,Z 1166.342,A 0.000,B 0.000,C 90.000,E1 61.591} C_DIS
LIN {X 0.046,Y -270.376,Z 1166.323,A 0.000,B 0.000,C 90.000,E1 58.152} C_DIS
LIN {X -0.001,Y -258.369,Z 1166.304,A 0.000,B 0.000,C 90.000,E1 54.642} C_DIS
LIN {X -0.035,Y -248.258,Z 1166.286,A 0.000,B 0.000,C 90.000,E1 51.412} C_DIS
LIN {X 0.106,Y -238.864,Z 1166.267,A 0.000,B 0.000,C 90.000,E1 48.081} C_DIS
LIN {X 0.083,Y -229.229,Z 1166.246,A 0.000,B 0.000,C 90.000,E1 44.352} C_DIS
LIN {X 0.099,Y -220.393,Z 1166.225,A 0.000,B 0.000,C 90.000,E1 40.539} C_DIS
LIN {X 0.088,Y -212.284,Z 1166.204,A 0.000,B 0.000,C 90.000,E1 36.664} C_DIS
LIN {X -0.032,Y -204.916,Z 1166.182,A 0.000,B 0.000,C 90.000,E1 32.752} C_DIS
LIN {X -0.020,Y -198.179,Z 1166.160,A 0.000,B 0.000,C 90.000,E1 28.743} C_DIS
LIN {X 0.099,Y -192.308,Z 1166.137,A 0.000,B 0.000,C 90.000,E1 24.643} C_DIS
LIN {X 0.000,Y -187.337,Z 1166.114,A 0.000,B 0.000,C 90.000,E1 20.556} C_DIS
LIN {X 0.027,Y -183.351,Z 1166.091,A 0.000,B 0.000,C 90.000,E1 16.386} C_DIS
LIN {X -0.037,Y -179.851,Z 1166.063,A 0.000,B 0.000,C 90.000,E1 11.366} C_DIS
LIN {X -0.024,Y -177.477,Z 1166.025,A 0.000,B 0.000,C 90.000,E1 4.588} C_DIS
LIN {X 0.014,Y -178.872,Z 1165.969,A 0.000,B 0.000,C 90.000,E1 354.432} C_DIS
LIN {X 0.067,Y -181.806,Z 1165.941,A 0.000,B 0.000,C 90.000,E1 349.342} C_DIS
LIN {X -0.029,Y -185.291,Z 1165.918,A 0.000,B 0.000,C 90.000,E1 345.172} C_DIS
LIN {X 0.041,Y -189.674,Z 1165.894,A 0.000,B 0.000,C 90.000,E1 340.986} C_DIS
LIN {X 0.023,Y -194.833,Z 1165.872,A 0.000,B 0.000,C 90.000,E1 336.869} C_DIS
LIN {X 0.028,Y -200.695,Z 1165.849,A 0.000,B 0.000,C 90.000,E1 332.794} C_DIS
LIN {X -0.030,Y -207.316,Z 1165.827,A 0.000,B 0.000,C 90.000,E1 328.791} C_DIS
LIN {X 0.020,Y -214.625,Z 1165.805,A 0.000,B 0.000,C 90.000,E1 324.815} C_DIS
LIN {X -0.004,Y -221.153,Z 1165.787,A 0.000,B 0.000,C 90.000,E1 321.698} C_DIS
LIN {X 0.030,Y -228.779,Z 1165.770,A 0.000,B 0.000,C 90.000,E1 318.609} C_DIS
LIN {X -0.102,Y -238.505,Z 1165.751,A 0.000,B 0.000,C 90.000,E1 315.243} C_DIS
LIN {X 0.055,Y -248.285,Z 1165.735,A 0.000,B 0.000,C 90.000,E1 312.243} C_DIS
LIN {X 0.007,Y -260.663,Z 1165.717,A 0.000,B 0.000,C 90.000,E1 308.991} C_DIS
LIN {X 0.033,Y -271.164,Z 1165.703,A 0.000,B 0.000,C 90.000,E1 306.503} C_DIS
LIN {X 0.031,Y -282.732,Z 1165.689,A 0.000,B 0.000,C 90.000,E1 304.072} C_DIS
LIN {X 0.139,Y -297.546,Z 1165.674,A 0.000,B 0.000,C 90.000,E1 301.337} C_DIS
LIN {X -0.183,Y -309.561,Z 1165.663,A 0.000,B 0.000,C 90.000,E1 299.411} C_DIS
LIN {X -0.018,Y -322.618,Z 1165.652,A 0.000,B 0.000,C 90.000,E1 297.436} C_DIS
LIN {X -0.019,Y -337.111,Z 1165.642,A 0.000,B 0.000,C 90.000,E1 295.540} C_DIS
LIN {X 0.148,Y -355.379,Z 1165.630,A 0.000,B 0.000,C 90.000,E1 293.387} C_DIS
LIN {X 0.075,Y -368.592,Z 1165.622,A 0.000,B 0.000,C 90.000,E1 292.025} C_DIS
LIN {X 0.109,Y -387.578,Z 1165.613,A 0.000,B 0.000,C 90.000,E1 290.248} C_DIS
LIN {X -0.104,Y -401.063,Z 1165.606,A 0.000,B 0.000,C 90.000,E1 289.033} C_DIS
LIN {X 0.097,Y -411.450,Z 1165.600,A 0.000,B 0.000,C 90.000,E1 288.000} C_DIS
LIN {X -0.058,Y -421.665,Z 1165.594,A 0.000,B 0.000,C 90.000,E1 286.985} C_DIS
LIN {X -0.166,Y -429.105,Z 1165.590,A 0.000,B 0.000,C 90.000,E1 286.205} C_DIS
LIN {X 0.063,Y -436.188,Z 1165.585,A 0.000,B 0.000,C 90.000,E1 285.371} C_DIS
LIN {X -0.082,Y -442.634,Z 1165.581,A 0.000,B 0.000,C 90.000,E1 284.592} C_DIS
LIN {X 0.143,Y -448.322,Z 1165.577,A 0.000,B 0.000,C 90.000,E1 283.772} C_DIS
LIN {X -0.007,Y -453.355,Z 1165.572,A 0.000,B 0.000,C 90.000,E1 283.008} C_DIS
LIN {X -0.118,Y -457.747,Z 1165.568,A 0.000,B 0.000,C 90.000,E1 282.243} C_DIS
LIN {X -0.189,Y -461.513,Z 1165.564,A 0.000,B 0.000,C 90.000,E1 281.478} C_DIS
LIN {X 0.221,Y -464.760,Z 1165.559,A 0.000,B 0.000,C 90.000,E1 280.658} C_DIS
LIN {X -0.182,Y -466.691,Z 1165.557,A 0.000,B 0.000,C 90.000,E1 280.197} C_DIS
LIN {X -0.039,Y -468.402,Z 1165.554,A 0.000,B 0.000,C 90.000,E1 279.670} C_DIS
LIN {X 0.039,Y -469.908,Z 1165.551,A 0.000,B 0.000,C 90.000,E1 279.151} C_DIS
LIN {X 0.200,Y -471.165,Z 1165.548,A 0.000,B 0.000,C 90.000,E1 278.624} C_DIS
LIN {X -0.168,Y -472.146,Z 1165.545,A 0.000,B 0.000,C 90.000,E1 278.163} C_DIS
LIN {X -0.059,Y -472.830,Z 1165.542,A 0.000,B 0.000,C 90.000,E1 277.644} C_DIS
LIN {X 0.056,Y -473.150,Z 1165.540,A 0.000,B 0.000,C 90.000,E1 277.125} C_DIS
LIN {X 0.177,Y -473.088,Z 1165.537,A 0.000,B 0.000,C 90.000,E1 276.606} C_DIS
LIN {X -0.171,Y -472.604,Z 1165.534,A 0.000,B 0.000,C 90.000,E1 276.144} C_DIS
LIN {X -0.049,Y -471.696,Z 1165.531,A 0.000,B 0.000,C 90.000,E1 275.625} C_DIS
LIN {X 0.069,Y -470.328,Z 1165.528,A 0.000,B 0.000,C 90.000,E1 275.106} C_DIS
LIN {X 0.178,Y -468.498,Z 1165.526,A 0.000,B 0.000,C 90.000,E1 274.588} C_DIS
LIN {X -0.221,Y -466.074,Z 1165.523,A 0.000,B 0.000,C 90.000,E1 274.131} C_DIS
LIN {X -0.137,Y -462.976,Z 1165.520,A 0.000,B 0.000,C 90.000,E1 273.612} C_DIS
LIN {X -0.073,Y -459.099,Z 1165.517,A 0.000,B 0.000,C 90.000,E1 273.094} C_DIS
LIN {X 0.164,Y -456.805,Z 1165.516,A 0.000,B 0.000,C 90.000,E1 272.808} C_DIS
LIN {X -0.198,Y -451.383,Z 1165.513,A 0.000,B 0.000,C 90.000,E1 272.350} C_DIS
LIN {X -0.204,Y -445.155,Z 1165.510,A 0.000,B 0.000,C 90.000,E1 271.892} C_DIS
LIN {X -0.091,Y -438.393,Z 1165.508,A 0.000,B 0.000,C 90.000,E1 271.489} C_DIS
LIN {X 0.071,Y -431.386,Z 1165.506,A 0.000,B 0.000,C 90.000,E1 271.146} C_DIS
LIN {X 0.205,Y -424.381,Z 1165.505,A 0.000,B 0.000,C 90.000,E1 270.859} C_DIS
LIN {X -0.192,Y -417.349,Z 1165.504,A 0.000,B 0.000,C 90.000,E1 270.688} C_DIS
LIN {X -0.095,Y -406.179,Z 1165.502,A 0.000,B 0.000,C 90.000,E1 270.401} C_DIS
LIN {X 0.028,Y -392.401,Z 1165.501,A 0.000,B 0.000,C 90.000,E1 270.115} C_DIS
LIN {X 0.007,Y -384.109,Z 1165.500,A 0.000,B 0.000,C 90.000,E1 270.000} C_DIS
LIN {X -0.066,Y -376.669,Z 1165.500,A 0.000,B 0.000,C 90.000,E1 269.943} C_DIS
LIN {X 0.158,Y -372.096,Z 1165.500,A 0.000,B 0.000,C 90.000,E1 269.885} C_DIS
LIN {X 0.053,Y -181.542,Z 1165.500,A 0.000,B 0.000,C 90.000,E1 269.885} C_DIS
LIN {X 0.050,Y -180.803,Z 1165.471,A 0.000,B 0.000,C 90.000,E1 264.780} C_DIS
LIN {X -0.053,Y -178.904,Z 1165.443,A 0.000,B 0.000,C 90.000,E1 259.746} C_DIS
LIN {X 0.027,Y -175.947,Z 1165.415,A 0.000,B 0.000,C 90.000,E1 254.629} C_DIS
LIN {X -0.026,Y -175.409,Z 1165.410,A 0.000,B 0.000,C 90.000,E1 253.795} C_DIS
LIN {X -0.023,Y -172.174,Z 1165.386,A 0.000,B 0.000,C 90.000,E1 249.518} C_DIS
LIN {X 0.017,Y -171.644,Z 1165.381,A 0.000,B 0.000,C 90.000,E1 248.646} C_DIS
LIN {X 0.011,Y -167.867,Z 1165.357,A 0.000,B 0.000,C 90.000,E1 244.332} C_DIS
LIN {X -0.045,Y -166.601,Z 1165.348,A 0.000,B 0.000,C 90.000,E1 242.615} C_DIS
LIN {X -0.051,Y -162.590,Z 1165.323,A 0.000,B 0.000,C 90.000,E1 238.250} C_DIS
LIN {X -0.077,Y -161.274,Z 1165.314,A 0.000,B 0.000,C 90.000,E1 236.501} C_DIS
LIN {X -0.042,Y -157.274,Z 1165.289,A 0.000,B 0.000,C 90.000,E1 232.065} C_DIS
LIN {X -0.018,Y -155.993,Z 1165.279,A 0.000,B 0.000,C 90.000,E1 230.275} C_DIS
LIN {X -0.057,Y -152.250,Z 1165.254,A 0.000,B 0.000,C 90.000,E1 225.810} C_DIS
LIN {X -0.035,Y -150.490,Z 1165.239,A 0.000,B 0.000,C 90.000,E1 223.095} C_DIS
LIN {X -0.004,Y -147.214,Z 1165.214,A 0.000,B 0.000,C 90.000,E1 218.543} C_DIS
LIN {X -0.035,Y -145.235,Z 1165.194,A 0.000,B 0.000,C 90.000,E1 214.898} C_DIS
LIN {X 0.076,Y -142.358,Z 1165.163,A 0.000,B 0.000,C 90.000,E1 209.333} C_DIS
LIN {X 0.003,Y -141.745,Z 1165.153,A 0.000,B 0.000,C 90.000,E1 207.513} C_DIS
LIN {X -0.071,Y -139.491,Z 1165.117,A 0.000,B 0.000,C 90.000,E1 201.046} C_DIS
LIN {X -0.033,Y -138.993,Z 1165.101,A 0.000,B 0.000,C 90.000,E1 198.236} C_DIS
LIN {X 0.060,Y -138.336,Z 1165.055,A 0.000,B 0.000,C 90.000,E1 189.792} C_DIS
LIN {X -0.055,Y -139.416,Z 1165.008,A 0.000,B 0.000,C 90.000,E1 181.432} C_DIS
LIN {X -0.002,Y -141.333,Z 1164.972,A 0.000,B 0.000,C 90.000,E1 174.894} C_DIS
LIN {X -0.045,Y -142.689,Z 1164.956,A 0.000,B 0.000,C 90.000,E1 172.129} C_DIS
LIN {X 0.076,Y -145.052,Z 1164.931,A 0.000,B 0.000,C 90.000,E1 167.465} C_DIS
LIN {X 0.073,Y -147.677,Z 1164.910,A 0.000,B 0.000,C 90.000,E1 163.795} C_DIS
LIN {X -0.034,Y -150.322,Z 1164.890,A 0.000,B 0.000,C 90.000,E1 160.188} C_DIS
LIN {X 0.037,Y -153.738,Z 1164.870,A 0.000,B 0.000,C 90.000,E1 156.538} C_DIS
LIN {X 0.028,Y -157.151,Z 1164.850,A 0.000,B 0.000,C 90.000,E1 152.948} C_DIS
LIN {X -0.037,Y -161.300,Z 1164.830,A 0.000,B 0.000,C 90.000,E1 149.410} C_DIS
LIN {X -0.020,Y -164.416,Z 1164.815,A 0.000,B 0.000,C 90.000,E1 146.755} C_DIS
LIN {X -0.024,Y -169.099,Z 1164.796,A 0.000,B 0.000,C 90.000,E1 143.256} C_DIS
LIN {X -0.073,Y -171.655,Z 1164.786,A 0.000,B 0.000,C 90.000,E1 141.537} C_DIS
LIN {X -0.027,Y -176.619,Z 1164.767,A 0.000,B 0.000,C 90.000,E1 138.081} C_DIS
LIN {X 0.102,Y -180.917,Z 1164.753,A 0.000,B 0.000,C 90.000,E1 135.486} C_DIS
LIN {X -0.035,Y -186.334,Z 1164.734,A 0.000,B 0.000,C 90.000,E1 132.162} C_DIS
LIN {X 0.032,Y -190.968,Z 1164.720,A 0.000,B 0.000,C 90.000,E1 129.644} C_DIS
LIN {X -0.050,Y -196.740,Z 1164.702,A 0.000,B 0.000,C 90.000,E1 126.377} C_DIS
LIN {X -0.073,Y -201.057,Z 1164.690,A 0.000,B 0.000,C 90.000,E1 124.199} C_DIS
LIN {X -0.155,Y -310.714,Z 1164.690,A 0.000,B 0.000,C 90.000,E1 124.199} C_DIS
LIN {X 0.194,Y -311.715,Z 1164.690,A 0.000,B 0.000,C 90.000,E1 124.119} C_DIS
LIN {X 0.056,Y -316.906,Z 1164.688,A 0.000,B 0.000,C 90.000,E1 123.913} C_DIS
LIN {X -0.073,Y -320.021,Z 1164.687,A 0.000,B 0.000,C 90.000,E1 123.658} C_DIS
LIN {X -0.177,Y -323.674,Z 1164.684,A 0.000,B 0.000,C 90.000,E1 123.166} C_DIS
LIN {X -0.095,Y -325.265,Z 1164.682,A 0.000,B 0.000,C 90.000,E1 122.832} C_DIS
LIN {X -0.178,Y -339.857,Z 1164.661,A 0.000,B 0.000,C 90.000,E1 119.077} C_DIS
LIN {X 0.006,Y -352.320,Z 1164.646,A 0.000,B 0.000,C 90.000,E1 116.283} C_DIS
LIN {X -0.060,Y -366.282,Z 1164.631,A 0.000,B 0.000,C 90.000,E1 113.590} C_DIS
LIN {X 0.016,Y -380.055,Z 1164.618,A 0.000,B 0.000,C 90.000,E1 111.227} C_DIS
LIN {X 0.164,Y -395.209,Z 1164.605,A 0.000,B 0.000,C 90.000,E1 108.906} C_DIS
LIN {X 0.057,Y -411.852,Z 1164.593,A 0.000,B 0.000,C 90.000,E1 106.677} C_DIS
LIN {X 0.124,Y -430.102,Z 1164.581,A 0.000,B 0.000,C 90.000,E1 104.481} C_DIS
LIN {X -0.110,Y -449.814,Z 1164.569,A 0.000,B 0.000,C 90.000,E1 102.411} C_DIS
LIN {X -0.228,Y -470.085,Z 1164.558,A 0.000,B 0.000,C 90.000,E1 100.489} C_DIS
LIN {X -0.196,Y -472.006,Z 1164.557,A 0.000,B 0.000,C 90.000,E1 100.254} C_DIS
LIN {X 0.126,Y -473.594,Z 1164.555,A 0.000,B 0.000,C 90.000,E1 99.962} C_DIS
LIN {X -0.020,Y -474.783,Z 1164.554,A 0.000,B 0.000,C 90.000,E1 99.726} C_DIS
LIN {X 0.097,Y -476.227,Z 1164.551,A 0.000,B 0.000,C 90.000,E1 99.208} C_DIS
LIN {X -0.246,Y -476.636,Z 1164.548,A 0.000,B 0.000,C 90.000,E1 98.746} C_DIS
LIN {X -0.038,Y -476.080,Z 1164.546,A 0.000,B 0.000,C 90.000,E1 98.219} C_DIS
LIN {X 0.101,Y -474.471,Z 1164.543,A 0.000,B 0.000,C 90.000,E1 97.701} C_DIS
LIN {X -0.035,Y -473.187,Z 1164.542,A 0.000,B 0.000,C 90.000,E1 97.466} C_DIS
LIN {X -0.174,Y -462.419,Z 1164.533,A 0.000,B 0.000,C 90.000,E1 95.967} C_DIS
LIN {X -0.076,Y -448.112,Z 1164.522,A 0.000,B 0.000,C 90.000,E1 93.898} C_DIS
LIN {X -0.014,Y -431.378,Z 1164.507,A 0.000,B 0.000,C 90.000,E1 91.260} C_DIS
LIN {X -0.121,Y -417.378,Z 1164.494,A 0.000,B 0.000,C 90.000,E1 88.854} C_DIS
LIN {X 0.099,Y -407.122,Z 1164.483,A 0.000,B 0.000,C 90.000,E1 86.906} C_DIS
LIN {X 0.152,Y -396.721,Z 1164.472,A 0.000,B 0.000,C 90.000,E1 84.951} C_DIS
LIN {X 0.065,Y -383.415,Z 1164.458,A 0.000,B 0.000,C 90.000,E1 82.413} C_DIS
LIN {X 0.093,Y -374.472,Z 1164.448,A 0.000,B 0.000,C 90.000,E1 80.679} C_DIS
LIN {X 0.083,Y -365.229,Z 1164.439,A 0.000,B 0.000,C 90.000,E1 78.926} C_DIS
LIN {X -0.090,Y -355.728,Z 1164.429,A 0.000,B 0.000,C 90.000,E1 77.173} C_DIS
LIN {X 0.071,Y -345.999,Z 1164.419,A 0.000,B 0.000,C 90.000,E1 75.338} C_DIS
LIN {X -0.077,Y -333.068,Z 1164.405,A 0.000,B 0.000,C 90.000,E1 72.906} C_DIS
LIN {X -0.044,Y -317.426,Z 1164.387,A 0.000,B 0.000,C 90.000,E1 69.752} C_DIS
LIN {X 0.137,Y -302.835,Z 1164.370,A 0.000,B 0.000,C 90.000,E1 66.485} C_DIS
LIN {X -0.160,Y -291.798,Z 1164.355,A 0.000,B 0.000,C 90.000,E1 63.896} C_DIS
LIN {X -0.104,Y -279.907,Z 1164.338,A 0.000,B 0.000,C 90.000,E1 60.845} C_DIS
LIN {X 0.029,Y -268.651,Z 1164.321,A 0.000,B 0.000,C 90.000,E1 57.709} C_DIS
LIN {X -0.056,Y -256.731,Z 1164.301,A 0.000,B 0.000,C 90.000,E1 54.196} C_DIS
LIN {X 0.031,Y -246.670,Z 1164.283,A 0.000,B 0.000,C 90.000,E1 50.928} C_DIS
LIN {X 0.117,Y -236.432,Z 1164.263,A 0.000,B 0.000,C 90.000,E1 47.229} C_DIS
LIN {X 0.020,Y -226.978,Z 1164.242,A 0.000,B 0.000,C 90.000,E1 43.500} C_DIS
LIN {X 0.136,Y -218.304,Z 1164.220,A 0.000,B 0.000,C 90.000,E1 39.644} C_DIS
LIN {X -0.069,Y -210.310,Z 1164.199,A 0.000,B 0.000,C 90.000,E1 35.804} C_DIS
LIN {X 0.093,Y -203.071,Z 1164.177,A 0.000,B 0.000,C 90.000,E1 31.799} C_DIS
LIN {X -0.010,Y -197.729,Z 1164.159,A 0.000,B 0.000,C 90.000,E1 28.615} C_DIS
LIN {X 0.095,Y -191.869,Z 1164.136,A 0.000,B 0.000,C 90.000,E1 24.515} C_DIS
LIN {X -0.019,Y -186.913,Z 1164.113,A 0.000,B 0.000,C 90.000,E1 20.429} C_DIS
LIN {X -0.010,Y -182.947,Z 1164.090,A 0.000,B 0.000,C 90.000,E1 16.260} C_DIS
LIN {X -0.021,Y -179.943,Z 1164.067,A 0.000,B 0.000,C 90.000,E1 12.063} C_DIS
LIN {X -0.040,Y -177.474,Z 1164.034,A 0.000,B 0.000,C 90.000,E1 6.144} C_DIS
LIN {X 0.001,Y -178.531,Z 1163.969,A 0.000,B 0.000,C 90.000,E1 354.432} C_DIS
LIN {X 0.041,Y -181.466,Z 1163.941,A 0.000,B 0.000,C 90.000,E1 349.342} C_DIS
LIN {X -0.065,Y -184.941,Z 1163.917,A 0.000,B 0.000,C 90.000,E1 345.172} C_DIS
LIN {X 0.055,Y -189.308,Z 1163.894,A 0.000,B 0.000,C 90.000,E1 340.967} C_DIS
LIN {X -0.038,Y -194.461,Z 1163.871,A 0.000,B 0.000,C 90.000,E1 336.869} C_DIS
LIN {X -0.046,Y -200.323,Z 1163.849,A 0.000,B 0.000,C 90.000,E1 332.794} C_DIS
LIN {X 0.058,Y -206.954,Z 1163.826,A 0.000,B 0.000,C 90.000,E1 328.742} C_DIS
LIN {X -0.051,Y -212.767,Z 1163.809,A 0.000,B 0.000,C 90.000,E1 325.595} C_DIS
LIN {X 0.051,Y -219.115,Z 1163.791,A 0.000,B 0.000,C 90.000,E1 322.431} C_DIS
LIN {X -0.114,Y -226.514,Z 1163.774,A 0.000,B 0.000,C 90.000,E1 319.380} C_DIS
LIN {X -0.154,Y -236.064,Z 1163.755,A 0.000,B 0.000,C 90.000,E1 315.972} C_DIS
LIN {X 0.102,Y -245.613,Z 1163.739,A 0.000,B 0.000,C 90.000,E1 312.933} C_DIS
LIN {X 0.091,Y -254.909,Z 1163.724,A 0.000,B 0.000,C 90.000,E1 310.378} C_DIS
LIN {X 0.108,Y -268.018,Z 1163.707,A 0.000,B 0.000,C 90.000,E1 307.156} C_DIS
LIN {X -0.088,Y -281.033,Z 1163.691,A 0.000,B 0.000,C 90.000,E1 304.405} C_DIS
LIN {X -0.025,Y -293.793,Z 1163.678,A 0.000,B 0.000,C 90.000,E1 302.005} C_DIS
LIN {X 0.024,Y -307.581,Z 1163.665,A 0.000,B 0.000,C 90.000,E1 299.667} C_DIS
LIN {X 0.077,Y -322.771,Z 1163.652,A 0.000,B 0.000,C 90.000,E1 297.385} C_DIS
LIN {X -0.166,Y -334.701,Z 1163.643,A 0.000,B 0.000,C 90.000,E1 295.848} C_DIS
LIN {X -0.059,Y -355.487,Z 1163.630,A 0.000,B 0.000,C 90.000,E1 293.387} C_DIS
LIN {X -0.118,Y -371.356,Z 1163.621,A 0.000,B 0.000,C 90.000,E1 291.770} C_DIS
LIN {X 0.023,Y -387.551,Z 1163.613,A 0.000,B 0.000,C 90.000,E1 290.248} C_DIS
LIN {X -0.085,Y -398.413,Z 1163.607,A 0.000,B 0.000,C 90.000,E1 289.268} C_DIS
LIN {X 0.162,Y -408.871,Z 1163.601,A 0.000,B 0.000,C 90.000,E1 288.236} C_DIS
LIN {X 0.180,Y -418.972,Z 1163.596,A 0.000,B 0.000,C 90.000,E1 287.221} C_DIS
LIN {X 0.157,Y -426.490,Z 1163.591,A 0.000,B 0.000,C 90.000,E1 286.441} C_DIS
LIN {X -0.024,Y -433.739,Z 1163.587,A 0.000,B 0.000,C 90.000,E1 285.662} C_DIS
LIN {X 0.226,Y -440.462,Z 1163.583,A 0.000,B 0.000,C 90.000,E1 284.828} C_DIS
LIN {X 0.007,Y -446.413,Z 1163.578,A 0.000,B 0.000,C 90.000,E1 284.064} C_DIS
LIN {X -0.168,Y -451.713,Z 1163.574,A 0.000,B 0.000,C 90.000,E1 283.300} C_DIS
LIN {X 0.154,Y -456.331,Z 1163.569,A 0.000,B 0.000,C 90.000,E1 282.479} C_DIS
LIN {X 0.070,Y -460.295,Z 1163.565,A 0.000,B 0.000,C 90.000,E1 281.715} C_DIS
LIN {X 0.021,Y -463.712,Z 1163.561,A 0.000,B 0.000,C 90.000,E1 280.950} C_DIS
LIN {X -0.091,Y -466.737,Z 1163.557,A 0.000,B 0.000,C 90.000,E1 280.197} C_DIS
LIN {X 0.053,Y -468.453,Z 1163.554,A 0.000,B 0.000,C 90.000,E1 279.670} C_DIS
LIN {X 0.131,Y -469.963,Z 1163.551,A 0.000,B 0.000,C 90.000,E1 279.151} C_DIS
LIN {X -0.172,Y -471.285,Z 1163.548,A 0.000,B 0.000,C 90.000,E1 278.681} C_DIS
LIN {X -0.074,Y -472.297,Z 1163.545,A 0.000,B 0.000,C 90.000,E1 278.163} C_DIS
LIN {X 0.035,Y -472.966,Z 1163.542,A 0.000,B 0.000,C 90.000,E1 277.644} C_DIS
LIN {X 0.151,Y -473.354,Z 1163.540,A 0.000,B 0.000,C 90.000,E1 277.125} C_DIS
LIN {X -0.198,Y -473.338,Z 1163.537,A 0.000,B 0.000,C 90.000,E1 276.663} C_DIS
LIN {X -0.074,Y -472.896,Z 1163.534,A 0.000,B 0.000,C 90.000,E1 276.144} C_DIS
LIN {X 0.049,Y -471.994,Z 1163.531,A 0.000,B 0.000,C 90.000,E1 275.625} C_DIS
LIN {X 0.168,Y -470.666,Z 1163.528,A 0.000,B 0.000,C 90.000,E1 275.106} C_DIS
LIN {X -0.188,Y -468.845,Z 1163.526,A 0.000,B 0.000,C 90.000,E1 274.645} C_DIS
LIN {X -0.120,Y -466.499,Z 1163.523,A 0.000,B 0.000,C 90.000,E1 274.131} C_DIS
LIN {X -0.034,Y -463.473,Z 1163.520,A 0.000,B 0.000,C 90.000,E1 273.612} C_DIS
LIN {X 0.032,Y -459.634,Z 1163.517,A 0.000,B 0.000,C 90.000,E1 273.094} C_DIS
LIN {X -0.186,Y -457.377,Z 1163.516,A 0.000,B 0.000,C 90.000,E1 272.865} C_DIS
LIN {X -0.096,Y -452.008,Z 1163.513,A 0.000,B 0.000,C 90.000,E1 272.350} C_DIS
LIN {X 0.206,Y -448.901,Z 1163.512,A 0.000,B 0.000,C 90.000,E1 272.064} C_DIS
LIN {X -0.140,Y -445.833,Z 1163.510,A 0.000,B 0.000,C 90.000,E1 271.892} C_DIS
LIN {X -0.062,Y -439.156,Z 1163.508,A 0.000,B 0.000,C 90.000,E1 271.489} C_DIS
LIN {X 0.096,Y -432.222,Z 1163.506,A 0.000,B 0.000,C 90.000,E1 271.146} C_DIS
LIN {X -0.209,Y -425.248,Z 1163.505,A 0.000,B 0.000,C 90.000,E1 270.917} C_DIS
LIN {X 0.209,Y -418.184,Z 1163.504,A 0.000,B 0.000,C 90.000,E1 270.630} C_DIS
LIN {X 0.045,Y -410.761,Z 1163.503,A 0.000,B 0.000,C 90.000,E1 270.458} C_DIS
LIN {X -0.003,Y -396.710,Z 1163.501,A 0.000,B 0.000,C 90.000,E1 270.172} C_DIS
LIN {X -0.070,Y -389.625,Z 1163.500,A 0.000,B 0.000,C 90.000,E1 270.057} C_DIS
LIN {X -0.013,Y -380.397,Z 1163.500,A 0.000,B 0.000,C 90.000,E1 269.943} C_DIS
LIN {X 0.056,Y -372.215,Z 1163.499,A 0.000,B 0.000,C 90.000,E1 269.885} C_DIS
LIN {X 0.004,Y -181.539,Z 1163.499,A 0.000,B 0.000,C 90.000,E1 269.885} C_DIS
LIN {X 0.004,Y -180.799,Z 1163.471,A 0.000,B 0.000,C 90.000,E1 264.780} C_DIS
LIN {X 0.078,Y -178.898,Z 1163.443,A 0.000,B 0.000,C 90.000,E1 259.690} C_DIS
LIN {X -0.017,Y -175.941,Z 1163.415,A 0.000,B 0.000,C 90.000,E1 254.629} C_DIS
LIN {X -0.071,Y -175.395,Z 1163.410,A 0.000,B 0.000,C 90.000,E1 253.795} C_DIS
LIN {X -0.067,Y -172.165,Z 1163.386,A 0.000,B 0.000,C 90.000,E1 249.518} C_DIS
LIN {X -0.027,Y -171.633,Z 1163.381,A 0.000,B 0.000,C 90.000,E1 248.646} C_DIS
LIN {X -0.033,Y -167.856,Z 1163.357,A 0.000,B 0.000,C 90.000,E1 244.332} C_DIS
LIN {X -0.089,Y -166.588,Z 1163.348,A 0.000,B 0.000,C 90.000,E1 242.615} C_DIS
LIN {X 0.045,Y -162.578,Z 1163.323,A 0.000,B 0.000,C 90.000,E1 238.201} C_DIS
LIN {X 0.104,Y -161.261,Z 1163.314,A 0.000,B 0.000,C 90.000,E1 236.421} C_DIS
LIN {X 0.013,Y -157.262,Z 1163.289,A 0.000,B 0.000,C 90.000,E1 232.029} C_DIS
LIN {X -0.060,Y -155.983,Z 1163.279,A 0.000,B 0.000,C 90.000,E1 230.275} C_DIS
LIN {X -0.099,Y -152.239,Z 1163.254,A 0.000,B 0.000,C 90.000,E1 225.810} C_DIS
LIN {X 0.027,Y -150.480,Z 1163.239,A 0.000,B 0.000,C 90.000,E1 223.056} C_DIS
LIN {X -0.045,Y -147.204,Z 1163.214,A 0.000,B 0.000,C 90.000,E1 218.543} C_DIS
LIN {X -0.074,Y -145.225,Z 1163.194,A 0.000,B 0.000,C 90.000,E1 214.898} C_DIS
LIN {X 0.036,Y -142.352,Z 1163.163,A 0.000,B 0.000,C 90.000,E1 209.333} C_DIS
LIN {X -0.036,Y -141.739,Z 1163.153,A 0.000,B 0.000,C 90.000,E1 207.513} C_DIS
LIN {X 0.071,Y -139.488,Z 1163.117,A 0.000,B 0.000,C 90.000,E1 200.972} C_DIS
LIN {X 0.060,Y -138.989,Z 1163.101,A 0.000,B 0.000,C 90.000,E1 198.181} C_DIS
LIN {X 0.021,Y -138.335,Z 1163.054,A 0.000,B 0.000,C 90.000,E1 189.792} C_DIS
LIN {X 0.045,Y -139.420,Z 1163.008,A 0.000,B 0.000,C 90.000,E1 181.375} C_DIS
LIN {X -0.041,Y -141.341,Z 1162.972,A 0.000,B 0.000,C 90.000,E1 174.894} C_DIS
LIN {X 0.076,Y -142.696,Z 1162.956,A 0.000,B 0.000,C 90.000,E1 172.064} C_DIS
LIN {X 0.036,Y -145.062,Z 1162.930,A 0.000,B 0.000,C 90.000,E1 167.465} C_DIS
LIN {X 0.033,Y -147.688,Z 1162.910,A 0.000,B 0.000,C 90.000,E1 163.795} C_DIS
LIN {X -0.075,Y -150.335,Z 1162.890,A 0.000,B 0.000,C 90.000,E1 160.188} C_DIS
LIN {X -0.004,Y -153.753,Z 1162.870,A 0.000,B 0.000,C 90.000,E1 156.538} C_DIS
LIN {X -0.013,Y -157.166,Z 1162.850,A 0.000,B 0.000,C 90.000,E1 152.948} C_DIS
LIN {X -0.079,Y -161.321,Z 1162.830,A 0.000,B 0.000,C 90.000,E1 149.410} C_DIS
LIN {X 0.075,Y -164.435,Z 1162.815,A 0.000,B 0.000,C 90.000,E1 146.707} C_DIS
LIN {X 0.068,Y -169.122,Z 1162.796,A 0.000,B 0.000,C 90.000,E1 143.210} C_DIS
LIN {X 0.017,Y -171.675,Z 1162.786,A 0.000,B 0.000,C 90.000,E1 141.492} C_DIS
LIN {X -0.073,Y -176.642,Z 1162.767,A 0.000,B 0.000,C 90.000,E1 138.081} C_DIS
LIN {X 0.055,Y -180.940,Z 1162.753,A 0.000,B 0.000,C 90.000,E1 135.486} C_DIS
LIN {X 0.043,Y -186.359,Z 1162.734,A 0.000,B 0.000,C 90.000,E1 132.123} C_DIS
LIN {X -0.016,Y -190.992,Z 1162.720,A 0.000,B 0.000,C 90.000,E1 129.644} C_DIS
LIN {X -0.098,Y -196.767,Z 1162.702,A 0.000,B 0.000,C 90.000,E1 126.377} C_DIS
LIN {X -0.031,Y -201.037,Z 1162.690,A 0.000,B 0.000,C 90.000,E1 124.199} C_DIS
LIN {X -0.095,Y -310.057,Z 1162.690,A 0.000,B 0.000,C 90.000,E1 124.199} C_DIS
LIN {X -0.143,Y -310.976,Z 1162.690,A 0.000,B 0.000,C 90.000,E1 124.199} C_DIS
LIN {X -0.019,Y -317.134,Z 1162.688,A 0.000,B 0.000,C 90.000,E1 123.913} C_DIS
LIN {X 0.090,Y -320.054,Z 1162.687,A 0.000,B 0.000,C 90.000,E1 123.627} C_DIS
LIN {X 0.202,Y -323.732,Z 1162.684,A 0.000,B 0.000,C 90.000,E1 123.086} C_DIS
LIN {X 0.011,Y -325.302,Z 1162.682,A 0.000,B 0.000,C 90.000,E1 122.801} C_DIS
LIN {X 0.070,Y -338.590,Z 1162.663,A 0.000,B 0.000,C 90.000,E1 119.333} C_DIS
LIN {X 0.071,Y -350.896,Z 1162.648,A 0.000,B 0.000,C 90.000,E1 116.565} C_DIS
LIN {X -0.208,Y -364.695,Z 1162.633,A 0.000,B 0.000,C 90.000,E1 113.898} C_DIS
LIN {X -0.179,Y -378.310,Z 1162.620,A 0.000,B 0.000,C 90.000,E1 111.535} C_DIS
LIN {X -0.081,Y -393.293,Z 1162.607,A 0.000,B 0.000,C 90.000,E1 109.214} C_DIS
LIN {X -0.121,Y -409.752,Z 1162.594,A 0.000,B 0.000,C 90.000,E1 106.968} C_DIS
LIN {X -0.123,Y -427.802,Z 1162.582,A 0.000,B 0.000,C 90.000,E1 104.773} C_DIS
LIN {X -0.064,Y -447.397,Z 1162.570,A 0.000,B 0.000,C 90.000,E1 102.647} C_DIS
LIN {X 0.154,Y -470.139,Z 1162.558,A 0.000,B 0.000,C 90.000,E1 100.433} C_DIS
LIN {X 0.189,Y -472.025,Z 1162.557,A 0.000,B 0.000,C 90.000,E1 100.197} C_DIS
LIN {X 0.045,Y -473.588,Z 1162.555,A 0.000,B 0.000,C 90.000,E1 99.962} C_DIS
LIN {X -0.100,Y -474.757,Z 1162.554,A 0.000,B 0.000,C 90.000,E1 99.726} C_DIS
LIN {X 0.017,Y -476.169,Z 1162.551,A 0.000,B 0.000,C 90.000,E1 99.208} C_DIS
LIN {X 0.145,Y -476.551,Z 1162.548,A 0.000,B 0.000,C 90.000,E1 98.690} C_DIS
LIN {X -0.119,Y -475.967,Z 1162.546,A 0.000,B 0.000,C 90.000,E1 98.219} C_DIS
LIN {X 0.021,Y -474.326,Z 1162.543,A 0.000,B 0.000,C 90.000,E1 97.701} C_DIS
LIN {X -0.115,Y -473.020,Z 1162.541,A 0.000,B 0.000,C 90.000,E1 97.466} C_DIS
LIN {X -0.190,Y -458.678,Z 1162.530,A 0.000,B 0.000,C 90.000,E1 95.448} C_DIS
LIN {X 0.193,Y -441.118,Z 1162.516,A 0.000,B 0.000,C 90.000,E1 92.808} C_DIS
LIN {X 0.171,Y -423.270,Z 1162.500,A 0.000,B 0.000,C 90.000,E1 89.885} C_DIS
LIN {X -0.058,Y -408.473,Z 1162.484,A 0.000,B 0.000,C 90.000,E1 87.192} C_DIS
LIN {X -0.006,Y -398.070,Z 1162.474,A 0.000,B 0.000,C 90.000,E1 85.241} C_DIS
LIN {X -0.100,Y -386.204,Z 1162.461,A 0.000,B 0.000,C 90.000,E1 82.996} C_DIS
LIN {X 0.035,Y -377.335,Z 1162.451,A 0.000,B 0.000,C 90.000,E1 81.254} C_DIS
LIN {X 0.014,Y -368.157,Z 1162.442,A 0.000,B 0.000,C 90.000,E1 79.511} C_DIS
LIN {X -0.103,Y -358.710,Z 1162.432,A 0.000,B 0.000,C 90.000,E1 77.757} C_DIS
LIN {X 0.031,Y -349.044,Z 1162.422,A 0.000,B 0.000,C 90.000,E1 75.936} C_DIS
LIN {X 0.060,Y -337.670,Z 1162.410,A 0.000,B 0.000,C 90.000,E1 73.795} C_DIS
LIN {X -0.093,Y -324.919,Z 1162.396,A 0.000,B 0.000,C 90.000,E1 71.329} C_DIS
LIN {X 0.100,Y -309.787,Z 1162.378,A 0.000,B 0.000,C 90.000,E1 68.103} C_DIS
LIN {X -0.004,Y -297.076,Z 1162.362,A 0.000,B 0.000,C 90.000,E1 65.177} C_DIS
LIN {X 0.053,Y -284.918,Z 1162.345,A 0.000,B 0.000,C 90.000,E1 62.153} C_DIS
LIN {X -0.017,Y -272.126,Z 1162.326,A 0.000,B 0.000,C 90.000,E1 58.742} C_DIS
LIN {X 0.042,Y -262.348,Z 1162.311,A 0.000,B 0.000,C 90.000,E1 55.928} C_DIS
LIN {X 0.053,Y -250.836,Z 1162.291,A 0.000,B 0.000,C 90.000,E1 52.351} C_DIS
LIN {X 0.091,Y -240.151,Z 1162.271,A 0.000,B 0.000,C 90.000,E1 48.690} C_DIS
LIN {X -0.051,Y -230.462,Z 1162.250,A 0.000,B 0.000,C 90.000,E1 45.000} C_DIS
LIN {X -0.008,Y -221.464,Z 1162.229,A 0.000,B 0.000,C 90.000,E1 41.191} C_DIS
LIN {X 0.012,Y -213.172,Z 1162.207,A 0.000,B 0.000,C 90.000,E1 37.317} C_DIS
LIN {X 0.041,Y -205.594,Z 1162.185,A 0.000,B 0.000,C 90.000,E1 33.372} C_DIS
LIN {X -0.097,Y -198.707,Z 1162.163,A 0.000,B 0.000,C 90.000,E1 29.411} C_DIS
LIN {X -0.042,Y -192.674,Z 1162.141,A 0.000,B 0.000,C 90.000,E1 25.335} C_DIS
LIN {X 0.036,Y -188.444,Z 1162.122,A 0.000,B 0.000,C 90.000,E1 22.025} C_DIS
LIN {X 0.034,Y -184.089,Z 1162.099,A 0.000,B 0.000,C 90.000,E1 17.873} C_DIS
LIN {X -0.031,Y -180.676,Z 1162.076,A 0.000,B 0.000,C 90.000,E1 13.703} C_DIS
LIN {X 0.058,Y -177.671,Z 1162.043,A 0.000,B 0.000,C 90.000,E1 7.757} C_DIS
LIN {X 0.026,Y -178.579,Z 1161.964,A 0.000,B 0.000,C 90.000,E1 353.571} C_DIS
LIN {X -0.058,Y -181.718,Z 1161.936,A 0.000,B 0.000,C 90.000,E1 348.522} C_DIS
LIN {X 0.066,Y -185.383,Z 1161.913,A 0.000,B 0.000,C 90.000,E1 344.283} C_DIS
LIN {X 0.017,Y -189.920,Z 1161.890,A 0.000,B 0.000,C 90.000,E1 340.134} C_DIS
LIN {X -0.100,Y -195.177,Z 1161.867,A 0.000,B 0.000,C 90.000,E1 336.049} C_DIS
LIN {X -0.088,Y -201.213,Z 1161.844,A 0.000,B 0.000,C 90.000,E1 331.975} C_DIS
LIN {X 0.068,Y -207.985,Z 1161.822,A 0.000,B 0.000,C 90.000,E1 327.916} C_DIS
LIN {X -0.039,Y -215.512,Z 1161.800,A 0.000,B 0.000,C 90.000,E1 323.989} C_DIS
LIN {X -0.087,Y -222.394,Z 1161.783,A 0.000,B 0.000,C 90.000,E1 320.884} C_DIS
LIN {X -0.017,Y -230.449,Z 1161.766,A 0.000,B 0.000,C 90.000,E1 317.796} C_DIS
LIN {X 0.088,Y -239.336,Z 1161.749,A 0.000,B 0.000,C 90.000,E1 314.757} C_DIS
LIN {X -0.073,Y -250.666,Z 1161.730,A 0.000,B 0.000,C 90.000,E1 311.472} C_DIS
LIN {X -0.063,Y -263.450,Z 1161.712,A 0.000,B 0.000,C 90.000,E1 308.222} C_DIS
LIN {X 0.074,Y -274.387,Z 1161.699,A 0.000,B 0.000,C 90.000,E1 305.724} C_DIS
LIN {X 0.032,Y -284.584,Z 1161.687,A 0.000,B 0.000,C 90.000,E1 303.658} C_DIS
LIN {X 0.193,Y -301.630,Z 1161.670,A 0.000,B 0.000,C 90.000,E1 300.590} C_DIS
LIN {X -0.057,Y -314.066,Z 1161.659,A 0.000,B 0.000,C 90.000,E1 298.665} C_DIS
LIN {X -0.036,Y -325.233,Z 1161.650,A 0.000,B 0.000,C 90.000,E1 297.052} C_DIS
LIN {X 0.081,Y -337.341,Z 1161.641,A 0.000,B 0.000,C 90.000,E1 295.463} C_DIS
LIN {X 0.075,Y -355.595,Z 1161.630,A 0.000,B 0.000,C 90.000,E1 293.334} C_DIS
LIN {X -0.125,Y -369.106,Z 1161.622,A 0.000,B 0.000,C 90.000,E1 291.972} C_DIS
LIN {X 0.122,Y -387.811,Z 1161.612,A 0.000,B 0.000,C 90.000,E1 290.194} C_DIS
LIN {X 0.144,Y -398.520,Z 1161.607,A 0.000,B 0.000,C 90.000,E1 289.214} C_DIS
LIN {X 0.001,Y -409.003,Z 1161.601,A 0.000,B 0.000,C 90.000,E1 288.236} C_DIS
LIN {X 0.043,Y -419.101,Z 1161.596,A 0.000,B 0.000,C 90.000,E1 287.221} C_DIS
LIN {X 0.010,Y -426.596,Z 1161.591,A 0.000,B 0.000,C 90.000,E1 286.441} C_DIS
LIN {X -0.180,Y -433.884,Z 1161.587,A 0.000,B 0.000,C 90.000,E1 285.662} C_DIS
LIN {X -0.231,Y -438.461,Z 1161.584,A 0.000,B 0.000,C 90.000,E1 285.134} C_DIS
LIN {X 0.063,Y -444.636,Z 1161.579,A 0.000,B 0.000,C 90.000,E1 284.300} C_DIS
LIN {X -0.120,Y -450.165,Z 1161.575,A 0.000,B 0.000,C 90.000,E1 283.536} C_DIS
LIN {X 0.182,Y -455.034,Z 1161.571,A 0.000,B 0.000,C 90.000,E1 282.715} C_DIS
LIN {X 0.091,Y -459.192,Z 1161.566,A 0.000,B 0.000,C 90.000,E1 281.951} C_DIS
LIN {X 0.030,Y -462.801,Z 1161.562,A 0.000,B 0.000,C 90.000,E1 281.186} C_DIS
LIN {X -0.245,Y -466.868,Z 1161.557,A 0.000,B 0.000,C 90.000,E1 280.197} C_DIS
LIN {X -0.100,Y -468.607,Z 1161.554,A 0.000,B 0.000,C 90.000,E1 279.670} C_DIS
LIN {X -0.022,Y -470.141,Z 1161.551,A 0.000,B 0.000,C 90.000,E1 279.151} C_DIS
LIN {X 0.141,Y -471.459,Z 1161.548,A 0.000,B 0.000,C 90.000,E1 278.624} C_DIS
LIN {X -0.226,Y -472.484,Z 1161.545,A 0.000,B 0.000,C 90.000,E1 278.163} C_DIS
LIN {X -0.116,Y -473.219,Z 1161.542,A 0.000,B 0.000,C 90.000,E1 277.644} C_DIS
LIN {X 0.001,Y -473.573,Z 1161.540,A 0.000,B 0.000,C 90.000,E1 277.125} C_DIS
LIN {X 0.124,Y -473.566,Z 1161.537,A 0.000,B 0.000,C 90.000,E1 276.606} C_DIS
LIN {X -0.222,Y -473.133,Z 1161.534,A 0.000,B 0.000,C 90.000,E1 276.144} C_DIS
LIN {X -0.096,Y -472.237,Z 1161.531,A 0.000,B 0.000,C 90.000,E1 275.625} C_DIS
LIN {X 0.024,Y -470.907,Z 1161.528,A 0.000,B 0.000,C 90.000,E1 275.106} C_DIS
LIN {X -0.063,Y -468.047,Z 1161.524,A 0.000,B 0.000,C 90.000,E1 274.359} C_DIS
LIN {X 0.032,Y -465.332,Z 1161.521,A 0.000,B 0.000,C 90.000,E1 273.841} C_DIS
LIN {X -0.171,Y -463.768,Z 1161.520,A 0.000,B 0.000,C 90.000,E1 273.612} C_DIS
LIN {X -0.102,Y -459.934,Z 1161.517,A 0.000,B 0.000,C 90.000,E1 273.094} C_DIS
LIN {X -0.079,Y -455.090,Z 1161.514,A 0.000,B 0.000,C 90.000,E1 272.579} C_DIS
LIN {X 0.196,Y -452.267,Z 1161.513,A 0.000,B 0.000,C 90.000,E1 272.293} C_DIS
LIN {X 0.126,Y -446.048,Z 1161.510,A 0.000,B 0.000,C 90.000,E1 271.835} C_DIS
LIN {X 0.193,Y -439.344,Z 1161.508,A 0.000,B 0.000,C 90.000,E1 271.432} C_DIS
LIN {X -0.090,Y -432.385,Z 1161.506,A 0.000,B 0.000,C 90.000,E1 271.146} C_DIS
LIN {X -0.027,Y -421.848,Z 1161.504,A 0.000,B 0.000,C 90.000,E1 270.745} C_DIS
LIN {X 0.053,Y -414.355,Z 1161.503,A 0.000,B 0.000,C 90.000,E1 270.516} C_DIS
LIN {X -0.064,Y -403.364,Z 1161.502,A 0.000,B 0.000,C 90.000,E1 270.286} C_DIS
LIN {X 0.154,Y -393.034,Z 1161.500,A 0.000,B 0.000,C 90.000,E1 270.057} C_DIS
LIN {X 0.138,Y -384.898,Z 1161.500,A 0.000,B 0.000,C 90.000,E1 269.943} C_DIS
LIN {X -0.020,Y -373.128,Z 1161.499,A 0.000,B 0.000,C 90.000,E1 269.885} C_DIS
LIN {X -0.058,Y -371.212,Z 1161.499,A 0.000,B 0.000,C 90.000,E1 269.885} C_DIS
LIN {X -0.046,Y -181.535,Z 1161.499,A 0.000,B 0.000,C 90.000,E1 269.885} C_DIS
LIN {X 0.080,Y -180.905,Z 1161.474,A 0.000,B 0.000,C 90.000,E1 265.298} C_DIS
LIN {X 0.030,Y -180.255,Z 1161.465,A 0.000,B 0.000,C 90.000,E1 263.628} C_DIS
LIN {X 0.049,Y -178.746,Z 1161.441,A 0.000,B 0.000,C 90.000,E1 259.398} C_DIS
LIN {X -0.054,Y -175.794,Z 1161.413,A 0.000,B 0.000,C 90.000,E1 254.338} C_DIS
LIN {X -0.059,Y -171.979,Z 1161.384,A 0.000,B 0.000,C 90.000,E1 249.209} C_DIS
LIN {X -0.020,Y -171.382,Z 1161.380,A 0.000,B 0.000,C 90.000,E1 248.337} C_DIS
LIN {X -0.035,Y -167.627,Z 1161.356,A 0.000,B 0.000,C 90.000,E1 244.024} C_DIS
LIN {X -0.020,Y -166.281,Z 1161.346,A 0.000,B 0.000,C 90.000,E1 242.281} C_DIS
LIN {X -0.026,Y -163.030,Z 1161.327,A 0.000,B 0.000,C 90.000,E1 238.791} C_DIS
LIN {X 0.026,Y -160.959,Z 1161.312,A 0.000,B 0.000,C 90.000,E1 236.135} C_DIS
LIN {X 0.011,Y -157.714,Z 1161.292,A 0.000,B 0.000,C 90.000,E1 232.603} C_DIS
LIN {X 0.073,Y -155.753,Z 1161.277,A 0.000,B 0.000,C 90.000,E1 229.908} C_DIS
LIN {X 0.019,Y -152.009,Z 1161.253,A 0.000,B 0.000,C 90.000,E1 225.445} C_DIS
LIN {X -0.071,Y -150.256,Z 1161.237,A 0.000,B 0.000,C 90.000,E1 222.771} C_DIS
LIN {X 0.063,Y -147.011,Z 1161.212,A 0.000,B 0.000,C 90.000,E1 218.177} C_DIS
LIN {X 0.053,Y -145.595,Z 1161.197,A 0.000,B 0.000,C 90.000,E1 215.438} C_DIS
LIN {X -0.027,Y -142.982,Z 1161.172,A 0.000,B 0.000,C 90.000,E1 210.875} C_DIS
LIN {X -0.027,Y -141.608,Z 1161.151,A 0.000,B 0.000,C 90.000,E1 207.180} C_DIS
LIN {X 0.015,Y -139.426,Z 1161.115,A 0.000,B 0.000,C 90.000,E1 200.663} C_DIS
LIN {X 0.065,Y -139.156,Z 1161.104,A 0.000,B 0.000,C 90.000,E1 198.779} C_DIS
LIN {X -0.048,Y -138.344,Z 1161.058,A 0.000,B 0.000,C 90.000,E1 190.423} C_DIS
LIN {X -0.067,Y -139.483,Z 1161.006,A 0.000,B 0.000,C 90.000,E1 181.088} C_DIS
LIN {X 0.014,Y -141.077,Z 1160.975,A 0.000,B 0.000,C 90.000,E1 175.469} C_DIS
LIN {X -0.033,Y -142.452,Z 1160.959,A 0.000,B 0.000,C 90.000,E1 172.704} C_DIS
LIN {X 0.058,Y -144.694,Z 1160.934,A 0.000,B 0.000,C 90.000,E1 168.049} C_DIS
LIN {X 0.010,Y -147.289,Z 1160.913,A 0.000,B 0.000,C 90.000,E1 164.393} C_DIS
LIN {X 0.026,Y -150.608,Z 1160.888,A 0.000,B 0.000,C 90.000,E1 159.826} C_DIS
LIN {X -0.038,Y -154.081,Z 1160.868,A 0.000,B 0.000,C 90.000,E1 156.230} C_DIS
LIN {X 0.027,Y -157.503,Z 1160.848,A 0.000,B 0.000,C 90.000,E1 152.615} C_DIS
LIN {X -0.028,Y -161.732,Z 1160.828,A 0.000,B 0.000,C 90.000,E1 149.076} C_DIS
LIN {X -0.015,Y -165.925,Z 1160.809,A 0.000,B 0.000,C 90.000,E1 145.548} C_DIS
LIN {X -0.028,Y -170.913,Z 1160.789,A 0.000,B 0.000,C 90.000,E1 142.065} C_DIS
LIN {X -0.001,Y -175.781,Z 1160.770,A 0.000,B 0.000,C 90.000,E1 138.609} C_DIS
LIN {X -0.001,Y -181.390,Z 1160.751,A 0.000,B 0.000,C 90.000,E1 135.202} C_DIS
LIN {X 0.003,Y -186.888,Z 1160.732,A 0.000,B 0.000,C 90.000,E1 131.838} C_DIS
LIN {X -0.045,Y -191.470,Z 1160.719,A 0.000,B 0.000,C 90.000,E1 129.358} C_DIS
LIN {X -0.113,Y -197.328,Z 1160.700,A 0.000,B 0.000,C 90.000,E1 126.091} C_DIS
LIN {X -0.050,Y -201.046,Z 1160.690,A 0.000,B 0.000,C 90.000,E1 124.199} C_DIS
LIN {X -0.125,Y -310.731,Z 1160.690,A 0.000,B 0.000,C 90.000,E1 124.199} C_DIS
LIN {X -0.015,Y -315.092,Z 1160.689,A 0.000,B 0.000,C 90.000,E1 124.040} C_DIS
LIN {X -0.079,Y -317.266,Z 1160.688,A 0.000,B 0.000,C 90.000,E1 123.913} C_DIS
LIN {X -0.031,Y -320.232,Z 1160.687,A 0.000,B 0.000,C 90.000,E1 123.627} C_DIS
LIN {X 0.024,Y -323.886,Z 1160.684,A 0.000,B 0.000,C 90.000,E1 123.086} C_DIS
LIN {X 0.108,Y -325.416,Z 1160.682,A 0.000,B 0.000,C 90.000,E1 122.752} C_DIS
LIN {X -0.111,Y -338.696,Z 1160.663,A 0.000,B 0.000,C 90.000,E1 119.333} C_DIS
LIN {X 0.043,Y -351.017,Z 1160.647,A 0.000,B 0.000,C 90.000,E1 116.539} C_DIS
LIN {X 0.084,Y -364.833,Z 1160.632,A 0.000,B 0.000,C 90.000,E1 113.823} C_DIS
LIN {X 0.119,Y -378.464,Z 1160.619,A 0.000,B 0.000,C 90.000,E1 111.461} C_DIS
LIN {X 0.223,Y -393.465,Z 1160.607,A 0.000,B 0.000,C 90.000,E1 109.141} C_DIS
LIN {X 0.071,Y -409.942,Z 1160.594,A 0.000,B 0.000,C 90.000,E1 106.913} C_DIS
LIN {X 0.087,Y -428.013,Z 1160.582,A 0.000,B 0.000,C 90.000,E1 104.717} C_DIS
LIN {X 0.170,Y -447.623,Z 1160.570,A 0.000,B 0.000,C 90.000,E1 102.591} C_DIS
LIN {X -0.040,Y -470.319,Z 1160.558,A 0.000,B 0.000,C 90.000,E1 100.433} C_DIS
LIN {X -0.004,Y -472.144,Z 1160.557,A 0.000,B 0.000,C 90.000,E1 100.197} C_DIS
LIN {X -0.148,Y -473.657,Z 1160.555,A 0.000,B 0.000,C 90.000,E1 99.962} C_DIS
LIN {X 0.175,Y -474.788,Z 1160.554,A 0.000,B 0.000,C 90.000,E1 99.670} C_DIS
LIN {X -0.175,Y -476.138,Z 1160.551,A 0.000,B 0.000,C 90.000,E1 99.208} C_DIS
LIN {X 0.025,Y -476.467,Z 1160.548,A 0.000,B 0.000,C 90.000,E1 98.681} C_DIS
LIN {X 0.160,Y -475.829,Z 1160.545,A 0.000,B 0.000,C 90.000,E1 98.163} C_DIS
LIN {X -0.172,Y -474.125,Z 1160.543,A 0.000,B 0.000,C 90.000,E1 97.701} C_DIS
LIN {X 0.161,Y -472.778,Z 1160.541,A 0.000,B 0.000,C 90.000,E1 97.409} C_DIS
LIN {X 0.074,Y -458.428,Z 1160.530,A 0.000,B 0.000,C 90.000,E1 95.391} C_DIS
LIN {X 0.002,Y -440.873,Z 1160.516,A 0.000,B 0.000,C 90.000,E1 92.808} C_DIS
LIN {X -0.022,Y -423.049,Z 1160.499,A 0.000,B 0.000,C 90.000,E1 89.885} C_DIS
LIN {X 0.159,Y -408.271,Z 1160.484,A 0.000,B 0.000,C 90.000,E1 87.135} C_DIS
LIN {X 0.162,Y -399.345,Z 1160.475,A 0.000,B 0.000,C 90.000,E1 85.469} C_DIS
LIN {X 0.049,Y -388.927,Z 1160.464,A 0.000,B 0.000,C 90.000,E1 83.514} C_DIS
LIN {X -0.174,Y -378.575,Z 1160.453,A 0.000,B 0.000,C 90.000,E1 81.546} C_DIS
LIN {X -0.169,Y -369.430,Z 1160.443,A 0.000,B 0.000,C 90.000,E1 79.803} C_DIS
LIN {X 0.119,Y -361.620,Z 1160.435,A 0.000,B 0.000,C 90.000,E1 78.285} C_DIS
LIN {X -0.041,Y -351.997,Z 1160.425,A 0.000,B 0.000,C 90.000,E1 76.520} C_DIS
LIN {X -0.032,Y -340.594,Z 1160.413,A 0.000,B 0.000,C 90.000,E1 74.393} C_DIS
LIN {X 0.097,Y -327.778,Z 1160.400,A 0.000,B 0.000,C 90.000,E1 71.891} C_DIS
LIN {X 0.064,Y -312.429,Z 1160.382,A 0.000,B 0.000,C 90.000,E1 68.720} C_DIS
LIN {X -0.075,Y -298.193,Z 1160.364,A 0.000,B 0.000,C 90.000,E1 65.485} C_DIS
LIN {X -0.116,Y -285.952,Z 1160.347,A 0.000,B 0.000,C 90.000,E1 62.487} C_DIS
LIN {X -0.093,Y -274.334,Z 1160.330,A 0.000,B 0.000,C 90.000,E1 59.410} C_DIS
LIN {X -0.121,Y -264.460,Z 1160.314,A 0.000,B 0.000,C 90.000,E1 56.628} C_DIS
LIN {X -0.036,Y -252.783,Z 1160.295,A 0.000,B 0.000,C 90.000,E1 53.050} C_DIS
LIN {X 0.094,Y -241.908,Z 1160.274,A 0.000,B 0.000,C 90.000,E1 49.380} C_DIS
LIN {X 0.011,Y -232.072,Z 1160.254,A 0.000,B 0.000,C 90.000,E1 45.688} C_DIS
LIN {X -0.053,Y -222.917,Z 1160.233,A 0.000,B 0.000,C 90.000,E1 41.919} C_DIS
LIN {X -0.012,Y -214.486,Z 1160.211,A 0.000,B 0.000,C 90.000,E1 38.051} C_DIS
LIN {X 0.052,Y -208.216,Z 1160.194,A 0.000,B 0.000,C 90.000,E1 34.898} C_DIS
LIN {X 0.033,Y -201.053,Z 1160.172,A 0.000,B 0.000,C 90.000,E1 30.924} C_DIS
LIN {X -0.040,Y -195.844,Z 1160.154,A 0.000,B 0.000,C 90.000,E1 27.719} C_DIS
LIN {X -0.071,Y -190.123,Z 1160.131,A 0.000,B 0.000,C 90.000,E1 23.643} C_DIS
LIN {X -0.061,Y -185.375,Z 1160.108,A 0.000,B 0.000,C 90.000,E1 19.504} C_DIS
LIN {X 0.016,Y -181.583,Z 1160.085,A 0.000,B 0.000,C 90.000,E1 15.300} C_DIS
LIN {X -0.027,Y -178.400,Z 1160.057,A 0.000,B 0.000,C 90.000,E1 10.254} C_DIS
LIN {X 0.059,Y -176.336,Z 1160.014,A 0.000,B 0.000,C 90.000,E1 2.579} C_DIS
LIN {X -0.022,Y -177.855,Z 1159.969,A 0.000,B 0.000,C 90.000,E1 354.432} C_DIS
LIN {X -0.008,Y -180.752,Z 1159.941,A 0.000,B 0.000,C 90.000,E1 349.342} C_DIS
LIN {X 0.041,Y -184.216,Z 1159.917,A 0.000,B 0.000,C 90.000,E1 345.117} C_DIS
LIN {X -0.042,Y -188.577,Z 1159.894,A 0.000,B 0.000,C 90.000,E1 340.967} C_DIS
LIN {X 0.094,Y -193.674,Z 1159.871,A 0.000,B 0.000,C 90.000,E1 336.794} C_DIS
LIN {X -0.019,Y -199.607,Z 1159.849,A 0.000,B 0.000,C 90.000,E1 332.743} C_DIS
LIN {X -0.100,Y -204.794,Z 1159.831,A 0.000,B 0.000,C 90.000,E1 329.537} C_DIS
LIN {X 0.042,Y -212.048,Z 1159.808,A 0.000,B 0.000,C 90.000,E1 325.515} C_DIS
LIN {X -0.043,Y -218.548,Z 1159.791,A 0.000,B 0.000,C 90.000,E1 322.396} C_DIS
LIN {X -0.045,Y -226.070,Z 1159.774,A 0.000,B 0.000,C 90.000,E1 319.299} C_DIS
LIN {X -0.086,Y -235.724,Z 1159.755,A 0.000,B 0.000,C 90.000,E1 315.891} C_DIS
LIN {X -0.015,Y -245.324,Z 1159.738,A 0.000,B 0.000,C 90.000,E1 312.894} C_DIS
LIN {X -0.017,Y -254.673,Z 1159.724,A 0.000,B 0.000,C 90.000,E1 310.334} C_DIS
LIN {X -0.002,Y -267.912,Z 1159.706,A 0.000,B 0.000,C 90.000,E1 307.111} C_DIS
LIN {X -0.092,Y -282.847,Z 1159.689,A 0.000,B 0.000,C 90.000,E1 303.992} C_DIS
LIN {X 0.012,Y -299.722,Z 1159.672,A 0.000,B 0.000,C 90.000,E1 300.924} C_DIS
LIN {X -0.006,Y -312.038,Z 1159.661,A 0.000,B 0.000,C 90.000,E1 298.949} C_DIS
LIN {X 0.066,Y -325.374,Z 1159.650,A 0.000,B 0.000,C 90.000,E1 297.001} C_DIS
LIN {X -0.088,Y -337.446,Z 1159.641,A 0.000,B 0.000,C 90.000,E1 295.463} C_DIS
LIN {X 0.044,Y -353.128,Z 1159.631,A 0.000,B 0.000,C 90.000,E1 293.590} C_DIS
LIN {X 0.219,Y -369.150,Z 1159.622,A 0.000,B 0.000,C 90.000,E1 291.897} C_DIS
LIN {X 0.031,Y -388.020,Z 1159.612,A 0.000,B 0.000,C 90.000,E1 290.174} C_DIS
LIN {X -0.175,Y -398.880,Z 1159.607,A 0.000,B 0.000,C 90.000,E1 289.214} C_DIS
LIN {X 0.037,Y -409.404,Z 1159.601,A 0.000,B 0.000,C 90.000,E1 288.181} C_DIS
LIN {X -0.138,Y -416.993,Z 1159.597,A 0.000,B 0.000,C 90.000,E1 287.457} C_DIS
LIN {X 0.051,Y -427.015,Z 1159.591,A 0.000,B 0.000,C 90.000,E1 286.386} C_DIS
LIN {X -0.062,Y -434.224,Z 1159.587,A 0.000,B 0.000,C 90.000,E1 285.607} C_DIS
LIN {X -0.168,Y -440.830,Z 1159.582,A 0.000,B 0.000,C 90.000,E1 284.828} C_DIS
LIN {X 0.044,Y -446.789,Z 1159.578,A 0.000,B 0.000,C 90.000,E1 284.008} C_DIS
LIN {X -0.125,Y -452.100,Z 1159.573,A 0.000,B 0.000,C 90.000,E1 283.244} C_DIS
LIN {X -0.244,Y -456.685,Z 1159.569,A 0.000,B 0.000,C 90.000,E1 282.479} C_DIS
LIN {X 0.122,Y -460.668,Z 1159.565,A 0.000,B 0.000,C 90.000,E1 281.658} C_DIS
LIN {X 0.078,Y -464.108,Z 1159.561,A 0.000,B 0.000,C 90.000,E1 280.894} C_DIS
LIN {X -0.029,Y -467.081,Z 1159.556,A 0.000,B 0.000,C 90.000,E1 280.141} C_DIS
LIN {X 0.118,Y -468.806,Z 1159.553,A 0.000,B 0.000,C 90.000,E1 279.613} C_DIS
LIN {X 0.199,Y -470.342,Z 1159.551,A 0.000,B 0.000,C 90.000,E1 279.095} C_DIS
LIN {X -0.102,Y -471.678,Z 1159.548,A 0.000,B 0.000,C 90.000,E1 278.624} C_DIS
LIN {X 0.000,Y -472.677,Z 1159.545,A 0.000,B 0.000,C 90.000,E1 278.106} C_DIS
LIN {X 0.112,Y -473.444,Z 1159.542,A 0.000,B 0.000,C 90.000,E1 277.587} C_DIS
LIN {X -0.239,Y -473.798,Z 1159.539,A 0.000,B 0.000,C 90.000,E1 277.125} C_DIS
LIN {X -0.115,Y -473.814,Z 1159.537,A 0.000,B 0.000,C 90.000,E1 276.606} C_DIS
LIN {X 0.012,Y -473.357,Z 1159.534,A 0.000,B 0.000,C 90.000,E1 276.087} C_DIS
LIN {X 0.138,Y -472.484,Z 1159.531,A 0.000,B 0.000,C 90.000,E1 275.568} C_DIS
LIN {X -0.210,Y -471.122,Z 1159.528,A 0.000,B 0.000,C 90.000,E1 275.106} C_DIS
LIN {X -0.094,Y -469.334,Z 1159.525,A 0.000,B 0.000,C 90.000,E1 274.588} C_DIS
LIN {X -0.023,Y -466.979,Z 1159.523,A 0.000,B 0.000,C 90.000,E1 274.073} C_DIS
LIN {X 0.066,Y -463.989,Z 1159.520,A 0.000,B 0.000,C 90.000,E1 273.555} C_DIS
LIN {X 0.133,Y -460.054,Z 1159.517,A 0.000,B 0.000,C 90.000,E1 273.037} C_DIS
LIN {X -0.084,Y -457.834,Z 1159.516,A 0.000,B 0.000,C 90.000,E1 272.808} C_DIS
LIN {X 0.156,Y -455.276,Z 1159.514,A 0.000,B 0.000,C 90.000,E1 272.522} C_DIS
LIN {X -0.012,Y -452.466,Z 1159.513,A 0.000,B 0.000,C 90.000,E1 272.293} C_DIS
LIN {X -0.052,Y -446.280,Z 1159.510,A 0.000,B 0.000,C 90.000,E1 271.835} C_DIS
LIN {X 0.028,Y -439.607,Z 1159.508,A 0.000,B 0.000,C 90.000,E1 271.432} C_DIS
LIN {X 0.179,Y -432.642,Z 1159.506,A 0.000,B 0.000,C 90.000,E1 271.088} C_DIS
LIN {X -0.113,Y -425.687,Z 1159.505,A 0.000,B 0.000,C 90.000,E1 270.859} C_DIS
LIN {X -0.123,Y -418.583,Z 1159.503,A 0.000,B 0.000,C 90.000,E1 270.630} C_DIS
LIN {X 0.124,Y -411.160,Z 1159.502,A 0.000,B 0.000,C 90.000,E1 270.401} C_DIS
LIN {X 0.062,Y -396.893,Z 1159.501,A 0.000,B 0.000,C 90.000,E1 270.115} C_DIS
LIN {X 0.003,Y -389.445,Z 1159.500,A 0.000,B 0.000,C 90.000,E1 270.000} C_DIS
LIN {X 0.070,Y -379.356,Z 1159.499,A 0.000,B 0.000,C 90.000,E1 269.885} C_DIS
LIN {X -0.153,Y -369.508,Z 1159.499,A 0.000,B 0.000,C 90.000,E1 269.885} C_DIS
LIN {X 0.070,Y -181.531,Z 1159.499,A 0.000,B 0.000,C 90.000,E1 269.828} C_DIS
LIN {X 0.000,Y -180.904,Z 1159.474,A 0.000,B 0.000,C 90.000,E1 265.298} C_DIS
LIN {X -0.050,Y -180.244,Z 1159.464,A 0.000,B 0.000,C 90.000,E1 263.628} C_DIS
LIN {X -0.031,Y -178.731,Z 1159.441,A 0.000,B 0.000,C 90.000,E1 259.398} C_DIS
LIN {X 0.036,Y -175.779,Z 1159.413,A 0.000,B 0.000,C 90.000,E1 254.283} C_DIS
LIN {X 0.024,Y -171.963,Z 1159.384,A 0.000,B 0.000,C 90.000,E1 249.156} C_DIS
LIN {X 0.061,Y -171.358,Z 1159.380,A 0.000,B 0.000,C 90.000,E1 248.284} C_DIS
LIN {X 0.039,Y -167.608,Z 1159.355,A 0.000,B 0.000,C 90.000,E1 243.973} C_DIS
LIN {X 0.051,Y -166.253,Z 1159.346,A 0.000,B 0.000,C 90.000,E1 242.231} C_DIS
LIN {X 0.039,Y -163.009,Z 1159.326,A 0.000,B 0.000,C 90.000,E1 238.742} C_DIS
LIN {X -0.048,Y -160.931,Z 1159.312,A 0.000,B 0.000,C 90.000,E1 236.135} C_DIS
LIN {X 0.062,Y -157.692,Z 1159.292,A 0.000,B 0.000,C 90.000,E1 232.557} C_DIS
LIN {X -0.001,Y -155.731,Z 1159.277,A 0.000,B 0.000,C 90.000,E1 229.908} C_DIS
LIN {X 0.054,Y -151.990,Z 1159.252,A 0.000,B 0.000,C 90.000,E1 225.405} C_DIS
LIN {X 0.070,Y -150.235,Z 1159.237,A 0.000,B 0.000,C 90.000,E1 222.690} C_DIS
LIN {X -0.007,Y -146.995,Z 1159.212,A 0.000,B 0.000,C 90.000,E1 218.177} C_DIS
LIN {X -0.017,Y -145.580,Z 1159.197,A 0.000,B 0.000,C 90.000,E1 215.438} C_DIS
LIN {X -0.023,Y -142.969,Z 1159.171,A 0.000,B 0.000,C 90.000,E1 210.846} C_DIS
LIN {X 0.030,Y -141.595,Z 1159.151,A 0.000,B 0.000,C 90.000,E1 207.129} C_DIS
LIN {X -0.054,Y -139.421,Z 1159.115,A 0.000,B 0.000,C 90.000,E1 200.663} C_DIS
LIN {X -0.003,Y -139.148,Z 1159.104,A 0.000,B 0.000,C 90.000,E1 198.779} C_DIS
LIN {X 0.019,Y -138.346,Z 1159.058,A 0.000,B 0.000,C 90.000,E1 190.366} C_DIS
LIN {X 0.005,Y -139.487,Z 1159.006,A 0.000,B 0.000,C 90.000,E1 181.031} C_DIS
LIN {X -0.056,Y -141.088,Z 1158.975,A 0.000,B 0.000,C 90.000,E1 175.469} C_DIS
LIN {X 0.039,Y -142.466,Z 1158.959,A 0.000,B 0.000,C 90.000,E1 172.648} C_DIS
LIN {X -0.013,Y -144.711,Z 1158.934,A 0.000,B 0.000,C 90.000,E1 168.049} C_DIS
LIN {X -0.062,Y -147.310,Z 1158.913,A 0.000,B 0.000,C 90.000,E1 164.393} C_DIS
LIN {X -0.046,Y -150.631,Z 1158.888,A 0.000,B 0.000,C 90.000,E1 159.826} C_DIS
LIN {X 0.029,Y -154.107,Z 1158.868,A 0.000,B 0.000,C 90.000,E1 156.177} C_DIS
LIN {X -0.047,Y -157.531,Z 1158.848,A 0.000,B 0.000,C 90.000,E1 152.615} C_DIS
LIN {X -0.103,Y -161.767,Z 1158.828,A 0.000,B 0.000,C 90.000,E1 149.076} C_DIS
LIN {X 0.003,Y -165.959,Z 1158.808,A 0.000,B 0.000,C 90.000,E1 145.515} C_DIS
LIN {X -0.001,Y -170.952,Z 1158.789,A 0.000,B 0.000,C 90.000,E1 142.029} C_DIS
LIN {X 0.051,Y -175.821,Z 1158.770,A 0.000,B 0.000,C 90.000,E1 138.566} C_DIS
LIN {X 0.046,Y -181.428,Z 1158.751,A 0.000,B 0.000,C 90.000,E1 135.162} C_DIS
LIN {X -0.080,Y -186.933,Z 1158.732,A 0.000,B 0.000,C 90.000,E1 131.838} C_DIS
LIN {X -0.007,Y -191.511,Z 1158.718,A 0.000,B 0.000,C 90.000,E1 129.322} C_DIS
LIN {X 0.078,Y -197.376,Z 1158.700,A 0.000,B 0.000,C 90.000,E1 126.011} C_DIS
LIN {X -0.073,Y -201.057,Z 1158.690,A 0.000,B 0.000,C 90.000,E1 124.199} C_DIS
LIN {X -0.161,Y -310.842,Z 1158.690,A 0.000,B 0.000,C 90.000,E1 124.199} C_DIS
LIN {X 0.174,Y -311.872,Z 1158.690,A 0.000,B 0.000,C 90.000,E1 124.119} C_DIS
LIN {X 0.050,Y -317.513,Z 1158.688,A 0.000,B 0.000,C 90.000,E1 123.865} C_DIS
LIN {X 0.100,Y -320.398,Z 1158.687,A 0.000,B 0.000,C 90.000,E1 123.579} C_DIS
LIN {X 0.091,Y -324.049,Z 1158.684,A 0.000,B 0.000,C 90.000,E1 123.038} C_DIS
LIN {X -0.097,Y -325.542,Z 1158.682,A 0.000,B 0.000,C 90.000,E1 122.752} C_DIS
LIN {X -0.025,Y -338.821,Z 1158.663,A 0.000,B 0.000,C 90.000,E1 119.283} C_DIS
LIN {X 0.144,Y -351.160,Z 1158.647,A 0.000,B 0.000,C 90.000,E1 116.488} C_DIS
LIN {X -0.133,Y -364.996,Z 1158.632,A 0.000,B 0.000,C 90.000,E1 113.823} C_DIS
LIN {X -0.101,Y -378.645,Z 1158.619,A 0.000,B 0.000,C 90.000,E1 111.461} C_DIS
LIN {X -0.001,Y -393.665,Z 1158.606,A 0.000,B 0.000,C 90.000,E1 109.141} C_DIS
LIN {X -0.159,Y -410.165,Z 1158.594,A 0.000,B 0.000,C 90.000,E1 106.913} C_DIS
LIN {X -0.147,Y -428.259,Z 1158.582,A 0.000,B 0.000,C 90.000,E1 104.717} C_DIS
LIN {X -0.062,Y -447.886,Z 1158.570,A 0.000,B 0.000,C 90.000,E1 102.591} C_DIS
LIN {X -0.214,Y -468.197,Z 1158.559,A 0.000,B 0.000,C 90.000,E1 100.658} C_DIS
LIN {X -0.177,Y -470.526,Z 1158.558,A 0.000,B 0.000,C 90.000,E1 100.423} C_DIS
LIN {X -0.225,Y -472.287,Z 1158.557,A 0.000,B 0.000,C 90.000,E1 100.197} C_DIS
LIN {X 0.098,Y -473.753,Z 1158.555,A 0.000,B 0.000,C 90.000,E1 99.905} C_DIS
LIN {X -0.046,Y -474.844,Z 1158.554,A 0.000,B 0.000,C 90.000,E1 99.670} C_DIS
LIN {X 0.074,Y -476.133,Z 1158.551,A 0.000,B 0.000,C 90.000,E1 99.151} C_DIS
LIN {X -0.197,Y -476.408,Z 1158.548,A 0.000,B 0.000,C 90.000,E1 98.681} C_DIS
LIN {X -0.061,Y -475.714,Z 1158.545,A 0.000,B 0.000,C 90.000,E1 98.163} C_DIS
LIN {X 0.078,Y -473.944,Z 1158.542,A 0.000,B 0.000,C 90.000,E1 97.644} C_DIS
LIN {X -0.058,Y -472.553,Z 1158.541,A 0.000,B 0.000,C 90.000,E1 97.409} C_DIS
LIN {X -0.145,Y -458.155,Z 1158.530,A 0.000,B 0.000,C 90.000,E1 95.391} C_DIS
LIN {X 0.224,Y -440.602,Z 1158.516,A 0.000,B 0.000,C 90.000,E1 92.751} C_DIS
LIN {X -0.118,Y -421.271,Z 1158.498,A 0.000,B 0.000,C 90.000,E1 89.599} C_DIS
LIN {X -0.058,Y -408.040,Z 1158.484,A 0.000,B 0.000,C 90.000,E1 87.135} C_DIS
LIN {X -0.054,Y -399.109,Z 1158.475,A 0.000,B 0.000,C 90.000,E1 85.469} C_DIS
LIN {X -0.116,Y -387.196,Z 1158.462,A 0.000,B 0.000,C 90.000,E1 83.223} C_DIS
LIN {X 0.003,Y -376.819,Z 1158.451,A 0.000,B 0.000,C 90.000,E1 81.197} C_DIS
LIN {X -0.027,Y -367.616,Z 1158.441,A 0.000,B 0.000,C 90.000,E1 79.454} C_DIS
LIN {X -0.121,Y -359.748,Z 1158.433,A 0.000,B 0.000,C 90.000,E1 77.993} C_DIS
LIN {X 0.032,Y -350.041,Z 1158.423,A 0.000,B 0.000,C 90.000,E1 76.172} C_DIS
LIN {X 0.078,Y -338.646,Z 1158.411,A 0.000,B 0.000,C 90.000,E1 74.031} C_DIS
LIN {X -0.153,Y -325.885,Z 1158.398,A 0.000,B 0.000,C 90.000,E1 71.583} C_DIS
LIN {X 0.063,Y -310.658,Z 1158.380,A 0.000,B 0.000,C 90.000,E1 68.358} C_DIS
LIN {X 0.108,Y -297.904,Z 1158.364,A 0.000,B 0.000,C 90.000,E1 65.409} C_DIS
LIN {X 0.082,Y -286.988,Z 1158.349,A 0.000,B 0.000,C 90.000,E1 62.743} C_DIS
LIN {X 0.124,Y -275.290,Z 1158.332,A 0.000,B 0.000,C 90.000,E1 59.665} C_DIS
LIN {X -0.029,Y -265.365,Z 1158.316,A 0.000,B 0.000,C 90.000,E1 56.914} C_DIS
LIN {X 0.075,Y -253.607,Z 1158.296,A 0.000,B 0.000,C 90.000,E1 53.336} C_DIS
LIN {X 0.075,Y -243.706,Z 1158.278,A 0.000,B 0.000,C 90.000,E1 50.070} C_DIS
LIN {X 0.048,Y -233.693,Z 1158.258,A 0.000,B 0.000,C 90.000,E1 46.377} C_DIS
